KUKA KRL program: EPS_2_251806_MH48A_A_20260213065146.src

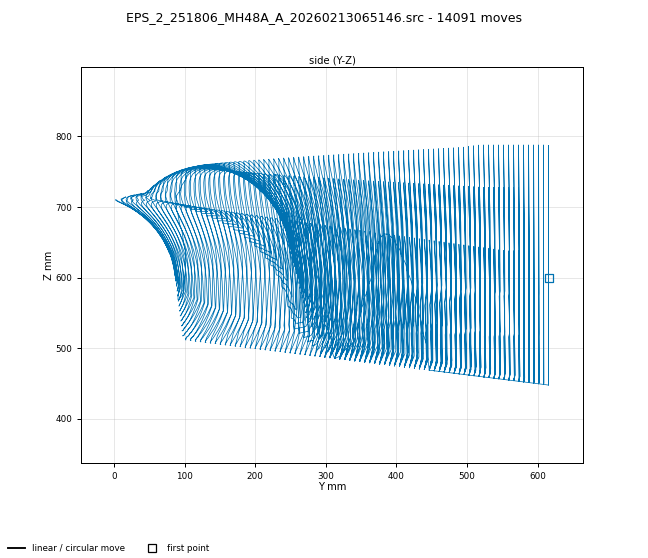
[picture p0: tool path of EPS_2_251806_MH48A_A_20260213065146.src, 14091 of 14093 moves have a stored position in this frame; points joined in program order, loops and branches not executed]
&ACCESS RVP
&REL 4
&COMMENT QRS 19112012
&PARAM EDITMASK = *
DEF PART()
EXT BAS (BAS_COMMAND :IN,REAL :IN )
INT I
BAS (#INITMOV,0 )

;KUKA QRS Post kuka4.cps  Date:22-06-2017 !

File_ID=3035

QRS_PRE_INIT()

;Init var - Until changes are made in qrs_pre_init
Outlet_Square_prg=0
Inlet_1_Square_prg=0
Inlet_2_Square_prg=0
Inlet_3_Square_prg=0
Inlet_4_Square_prg=0
Inlet_5_Square_prg=0

Outlet_1={X 0.000, Y 519.160, Z 687.500, B 0.000, E1 0.000 }
Inlet_1={X 0.000, Y 553.380, Z 207.500, B 0.000, E1 194.000 }
Inlet_2={X 0.000, Y 523.440, Z 627.500, B 0.000, E1 257.000 }
Outlet_1_type=201
Inlet_1_type=201
Inlet_2_type=201
;QRS#1=Sidecore dimensions
;QRS#2=200-8" PVC SDR 35
;QRS#3=200-8" PVC SDR 35
;QRS#4=200-8" PVC SDR 35
;QRS#5=
;QRS#6=
;QRS#7=
;QRS#8=
;QRS#9=12-08 PSX
;QRS#10=12-08 PSX
;QRS#11=12-08 PSX
;QRS#12=
;QRS#13=
;QRS#14=
;QRS#15=
;QRS#16=1220x127x1067 3,5'
;QRS#17=EPS Height
;QRS#18=788
;QRS#19=*
;QRS#20= UPDATED VERSION 22-06-2017
;QRS#21=*
Outlet_Square=0100
Inlet_1_Square=0100
Inlet_2_Square=0100
Inlet_3_Square=0
Inlet_4_Square=0
Inlet_5_Square=0
Mill_Square=1
Outlet_Square_Prg=204
Inlet_1_Square_prg=204
Inlet_2_Square_prg=204

QRS_INIT()

$ADVANCE=5

; T1
PTP {E1 173.589,E2 173.589}
PTP {X 0,Y 615.51,A -85,B 0,C 180,E1 173.589,E2 173.589,E3 0,E4 0,E5 0,E6 0}
QRS_SPEED_INIT()
LIN {X 0,Y 615.51,Z 600,A -85,B 0,C 180,E1 173.589,E2 173.589,E3 0,E4 0,E5 0,E6 0} C_VEL
LIN {X 0,Y 615.51,Z 457.871,A -85,B 0,C 180,E1 173.589,E2 173.589} C_VEL
LIN {X 0,Y 615.51,Z 449.702,A -85,B 0,C 180,E1 173.589,E2 173.589} C_VEL
LIN {X 0,Y 615.493,Z 447.702,A -85,B 0,C 180,E1 173.404,E2 173.404} C_VEL
LIN {X 0,Y 615.484,Z 447.686,A -85,B 0,C 180,E1 170.801,E2 170.801} C_VEL
LIN {X 0,Y 615.449,Z 447.691,A -85,B 0,C 180,E1 168.139,E2 168.139} C_VEL
LIN {X 0,Y 615.487,Z 447.699,A -85,B 0,C 180,E1 165.451,E2 165.451} C_VEL
LIN {X 0,Y 615.488,Z 447.685,A -85,B 0,C 180,E1 162.73,E2 162.73} C_VEL
LIN {X 0,Y 615.482,Z 447.685,A -85,B 0,C 180,E1 160.662,E2 160.662} C_VEL
LIN {X 0,Y 615.478,Z 447.685,A -85,B 0,C 180,E1 158.568,E2 158.568} C_VEL
LIN {X 0,Y 615.456,Z 447.69,A -85,B 0,C 180,E1 155.994,E2 155.994} C_VEL
LIN {X 0,Y 615.473,Z 447.695,A -85,B 0,C 180,E1 153.556,E2 153.556} C_VEL
LIN {X 0,Y 615.485,Z 447.685,A -85,B 0,C 180,E1 150.594,E2 150.594} C_VEL
LIN {X 0,Y 615.469,Z 447.686,A -85,B 0,C 180,E1 148.314,E2 148.314} C_VEL
LIN {X 0,Y 615.457,Z 447.689,A -85,B 0,C 180,E1 145.976,E2 145.976} C_VEL
LIN {X 0,Y 615.491,Z 447.698,A -85,B 0,C 180,E1 143.061,E2 143.061} C_VEL
LIN {X 0,Y 615.472,Z 447.685,A -85,B 0,C 180,E1 140.249,E2 140.249} C_VEL
LIN {X 0,Y 615.466,Z 447.692,A -85,B 0,C 180,E1 137.645,E2 137.645} C_VEL
LIN {X 0,Y 615.492,Z 447.695,A -85,B 0,C 180,E1 134.932,E2 134.932} C_VEL
LIN {X 0,Y 615.487,Z 447.683,A -85,B 0,C 180,E1 132.351,E2 132.351} C_VEL
LIN {X 0,Y 615.465,Z 447.689,A -85,B 0,C 180,E1 129.75,E2 129.75} C_VEL
LIN {X 0,Y 615.494,Z 447.697,A -85,B 0,C 180,E1 126.938,E2 126.938} C_VEL
LIN {X 0,Y 615.472,Z 447.685,A -85,B 0,C 180,E1 124.021,E2 124.021} C_VEL
LIN {X 0,Y 615.468,Z 447.688,A -85,B 0,C 180,E1 121.685,E2 121.685} C_VEL
LIN {X 0,Y 615.475,Z 447.692,A -85,B 0,C 180,E1 119.405,E2 119.405} C_VEL
LIN {X 0,Y 615.492,Z 447.685,A -85,B 0,C 180,E1 116.442,E2 116.442} C_VEL
LIN {X 0,Y 615.479,Z 447.683,A -85,B 0,C 180,E1 114.007,E2 114.007} C_VEL
LIN {X 0,Y 615.476,Z 447.69,A -85,B 0,C 180,E1 111.431,E2 111.431} C_VEL
LIN {X 0,Y 615.488,Z 447.691,A -85,B 0,C 180,E1 108.606,E2 108.606} C_VEL
LIN {X 0,Y 615.479,Z 447.683,A -85,B 0,C 180,E1 105.904,E2 105.904} C_VEL
LIN {X 0,Y 615.487,Z 447.692,A -85,B 0,C 180,E1 103.2,E2 103.2} C_VEL
LIN {X 0,Y 615.487,Z 447.691,A -85,B 0,C 180,E1 100.526,E2 100.526} C_VEL
LIN {X 0,Y 615.483,Z 447.682,A -85,B 0,C 180,E1 97.874,E2 97.874} C_VEL
LIN {X 0,Y 615.479,Z 447.691,A -85,B 0,C 180,E1 95.24,E2 95.24} C_VEL
LIN {X 0,Y 615.486,Z 447.696,A -85,B 0,C 180,E1 92.617,E2 92.617} C_VEL
LIN {X 0,Y 615.487,Z 447.682,A -85,B 0,C 180,E1 89.999,E2 89.999} C_VEL
LIN {X 0,Y 615.498,Z 447.858,A -85,B 0,C 180,E1 88.69,E2 88.69} C_VEL
LIN {X 0,Y 615.497,Z 448.887,A -85,B 0,C 180,E1 88.568,E2 88.568} C_VEL
LIN {X 0,Y 615.498,Z 534.909,A -85,B 0,C 180,E1 87.524,E2 87.524} C_VEL
LIN {X 0,Y 615.498,Z 548.363,A -85,B 0,C 180,E1 87.217,E2 87.217} C_VEL
LIN {X 0,Y 615.499,Z 560.522,A -85,B 0,C 180,E1 86.808,E2 86.808} C_VEL
LIN {X 0,Y 615.497,Z 571.457,A -85,B 0,C 180,E1 86.316,E2 86.316} C_VEL
LIN {X 0,Y 615.491,Z 582.851,A -85,B 0,C 180,E1 85.661,E2 85.661} C_VEL
LIN {X 0,Y 615.498,Z 593.126,A -85,B 0,C 180,E1 84.922,E2 84.922} C_VEL
LIN {X 0,Y 615.5,Z 602.443,A -85,B 0,C 180,E1 84.101,E2 84.101} C_VEL
LIN {X 0,Y 615.496,Z 611.559,A -85,B 0,C 180,E1 83.098,E2 83.098} C_VEL
LIN {X 0,Y 615.496,Z 618.714,A -85,B 0,C 180,E1 82.123,E2 82.123} C_VEL
LIN {X 0,Y 615.496,Z 624.559,A -85,B 0,C 180,E1 81.132,E2 81.132} C_VEL
LIN {X 0,Y 615.497,Z 629.171,A -85,B 0,C 180,E1 80.137,E2 80.137} C_VEL
LIN {X 0,Y 615.495,Z 632.785,A -85,B 0,C 180,E1 79.107,E2 79.107} C_VEL
LIN {X 0,Y 615.496,Z 635.187,A -85,B 0,C 180,E1 78.138,E2 78.138} C_VEL
LIN {X 0,Y 615.495,Z 636.338,A -85,B 0,C 180,E1 77.469,E2 77.469} C_VEL
LIN {X 0,Y 615.496,Z 637.354,A -85,B 0,C 180,E1 76.125,E2 76.125} C_VEL
LIN {X 0,Y 615.497,Z 637.271,A -85,B 0,C 180,E1 75.45,E2 75.45} C_VEL
LIN {X 0,Y 615.496,Z 636.73,A -85,B 0,C 180,E1 74.773,E2 74.773} C_VEL
LIN {X 0,Y 615.494,Z 634.742,A -85,B 0,C 180,E1 73.566,E2 73.566} C_VEL
LIN {X 0,Y 615.496,Z 631.451,A -85,B 0,C 180,E1 72.386,E2 72.386} C_VEL
LIN {X 0,Y 615.497,Z 627.367,A -85,B 0,C 180,E1 71.353,E2 71.353} C_VEL
LIN {X 0,Y 615.497,Z 620.936,A -85,B 0,C 180,E1 70.141,E2 70.141} C_VEL
LIN {X 0,Y 615.497,Z 613.795,A -85,B 0,C 180,E1 69.094,E2 69.094} C_VEL
LIN {X 0,Y 615.499,Z 606.395,A -85,B 0,C 180,E1 68.216,E2 68.216} C_VEL
LIN {X 0,Y 615.5,Z 598.08,A -85,B 0,C 180,E1 67.403,E2 67.403} C_VEL
LIN {X 0,Y 615.5,Z 588.295,A -85,B 0,C 180,E1 66.621,E2 66.621} C_VEL
LIN {X 0,Y 615.488,Z 577.552,A -85,B 0,C 180,E1 65.925,E2 65.925} C_VEL
LIN {X 0,Y 615.499,Z 565.779,A -85,B 0,C 180,E1 65.323,E2 65.323} C_VEL
LIN {X 0,Y 615.498,Z 553.895,A -85,B 0,C 180,E1 64.863,E2 64.863} C_VEL
LIN {X 0,Y 615.499,Z 540.76,A -85,B 0,C 180,E1 64.501,E2 64.501} C_VEL
LIN {X 0,Y 615.494,Z 528.044,A -85,B 0,C 180,E1 64.284,E2 64.284} C_VEL
LIN {X 0,Y 615.496,Z 449.024,A -85,B 0,C 180,E1 63.348,E2 63.348} C_VEL
LIN {X 0,Y 615.498,Z 447.914,A -85,B 0,C 180,E1 63.236,E2 63.236} C_VEL
LIN {X 0,Y 615.493,Z 447.694,A -85,B 0,C 180,E1 61.341,E2 61.341} C_VEL
LIN {X 0,Y 615.495,Z 447.693,A -85,B 0,C 180,E1 58.912,E2 58.912} C_VEL
LIN {X 0,Y 615.473,Z 447.687,A -85,B 0,C 180,E1 56.468,E2 56.468} C_VEL
LIN {X 0,Y 615.465,Z 447.687,A -85,B 0,C 180,E1 54.169,E2 54.169} C_VEL
LIN {X 0,Y 615.471,Z 447.686,A -85,B 0,C 180,E1 51.929,E2 51.929} C_VEL
LIN {X 0,Y 615.495,Z 447.692,A -85,B 0,C 180,E1 49.393,E2 49.393} C_VEL
LIN {X 0,Y 615.499,Z 447.687,A -85,B 0,C 180,E1 46.755,E2 46.755} C_VEL
LIN {X 0,Y 615.464,Z 447.688,A -85,B 0,C 180,E1 43.994,E2 43.994} C_VEL
LIN {X 0,Y 615.491,Z 447.699,A -85,B 0,C 180,E1 41.094,E2 41.094} C_VEL
LIN {X 0,Y 615.486,Z 447.694,A -85,B 0,C 180,E1 38.904,E2 38.904} C_VEL
LIN {X 0,Y 615.473,Z 447.686,A -85,B 0,C 180,E1 36.425,E2 36.425} C_VEL
LIN {X 0,Y 615.498,Z 447.832,A -85,B 0,C 180,E1 35.113,E2 35.113} C_VEL
LIN {X 0,Y 615.498,Z 452.891,A -85,B 0,C 180,E1 34.36,E2 34.36} C_VEL
LIN {X 0,Y 615.491,Z 473.395,A -85,B 0,C 180,E1 31.535,E2 31.535} C_VEL
LIN {X 0,Y 615.491,Z 494.595,A -85,B 0,C 180,E1 28.658,E2 28.658} C_VEL
LIN {X 0,Y 615.486,Z 515.486,A -85,B 0,C 180,E1 25.874,E2 25.874} C_VEL
LIN {X 0,Y 615.491,Z 517.349,A -85,B 0,C 180,E1 25.806,E2 25.806} C_VEL
LIN {X 0,Y 615.495,Z 624.013,A -85,B 0,C 180,E1 24.541,E2 24.541} C_VEL
LIN {X 0,Y 615.498,Z 637.597,A -85,B 0,C 180,E1 24.238,E2 24.238} C_VEL
LIN {X 0,Y 615.497,Z 649.703,A -85,B 0,C 180,E1 23.839,E2 23.839} C_VEL
LIN {X 0,Y 615.494,Z 661.987,A -85,B 0,C 180,E1 23.288,E2 23.288} C_VEL
LIN {X 0,Y 615.497,Z 673.863,A -85,B 0,C 180,E1 22.594,E2 22.594} C_VEL
LIN {X 0,Y 615.498,Z 683.775,A -85,B 0,C 180,E1 21.871,E2 21.871} C_VEL
LIN {X 0,Y 615.499,Z 692.646,A -85,B 0,C 180,E1 21.08,E2 21.08} C_VEL
LIN {X 0,Y 615.498,Z 701.024,A -85,B 0,C 180,E1 20.163,E2 20.163} C_VEL
LIN {X 0,Y 615.498,Z 708.439,A -85,B 0,C 180,E1 19.164,E2 19.164} C_VEL
LIN {X 0,Y 615.498,Z 713.741,A -85,B 0,C 180,E1 18.281,E2 18.281} C_VEL
LIN {X 0,Y 615.497,Z 718.599,A -85,B 0,C 180,E1 17.27,E2 17.27} C_VEL
LIN {X 0,Y 615.497,Z 721.746,A -85,B 0,C 180,E1 16.432,E2 16.432} C_VEL
LIN {X 0,Y 615.498,Z 724.997,A -85,B 0,C 180,E1 15.226,E2 15.226} C_VEL
LIN {X 0,Y 615.494,Z 726.224,A -85,B 0,C 180,E1 14.549,E2 14.549} C_VEL
LIN {X 0,Y 615.494,Z 726.988,A -85,B 0,C 180,E1 13.874,E2 13.874} C_VEL
LIN {X 0,Y 615.494,Z 727.294,A -85,B 0,C 180,E1 12.53,E2 12.53} C_VEL
LIN {X 0,Y 615.495,Z 726.833,A -85,B 0,C 180,E1 11.86,E2 11.86} C_VEL
LIN {X 0,Y 615.494,Z 725.432,A -85,B 0,C 180,E1 10.888,E2 10.888} C_VEL
LIN {X 0,Y 615.497,Z 721.911,A -85,B 0,C 180,E1 9.53,E2 9.53} C_VEL
LIN {X 0,Y 615.495,Z 718.153,A -85,B 0,C 180,E1 8.536,E2 8.536} C_VEL
LIN {X 0,Y 615.497,Z 713.28,A -85,B 0,C 180,E1 7.545,E2 7.545} C_VEL
LIN {X 0,Y 615.496,Z 707.158,A -85,B 0,C 180,E1 6.556,E2 6.556} C_VEL
LIN {X 0,Y 615.498,Z 699.562,A -85,B 0,C 180,E1 5.569,E2 5.569} C_VEL
LIN {X 0,Y 615.497,Z 690.049,A -85,B 0,C 180,E1 4.584,E2 4.584} C_VEL
LIN {X 0,Y 615.5,Z 680.271,A -85,B 0,C 180,E1 3.764,E2 3.764} C_VEL
LIN {X 0,Y 615.493,Z 669.27,A -85,B 0,C 180,E1 3.027,E2 3.027} C_VEL
LIN {X 0,Y 615.497,Z 658.558,A -85,B 0,C 180,E1 2.454,E2 2.454} C_VEL
LIN {X 0,Y 615.499,Z 646.783,A -85,B 0,C 180,E1 1.963,E2 1.963} C_VEL
LIN {X 0,Y 615.498,Z 634.795,A -85,B 0,C 180,E1 1.595,E2 1.595} C_VEL
LIN {X 0,Y 615.499,Z 622.775,A -85,B 0,C 180,E1 1.349,E2 1.349} C_VEL
LIN {X 0,Y 615.493,Z 516.279,A -85,B 0,C 180,E1 0.082,E2 0.082} C_VEL
LIN {X 0,Y 615.486,Z 515.176,A -85,B 0,C 180,E1 0,E2 0} C_VEL
LIN {X 0,Y 615.485,Z 494.453,A -85,B 0,C 180,E1 -2.782,E2 -2.782} C_VEL
LIN {X 0,Y 615.499,Z 473.986,A -85,B 0,C 180,E1 -5.57,E2 -5.57} C_VEL
LIN {X 0,Y 615.496,Z 453.734,A -85,B 0,C 180,E1 -8.371,E2 -8.371} C_VEL
LIN {X 0,Y 615.498,Z 447.975,A -85,B 0,C 180,E1 -9.199,E2 -9.199} C_VEL
LIN {X 0,Y 615.461,Z 447.692,A -85,B 0,C 180,E1 -9.863,E2 -9.863} C_VEL
LIN {X 0,Y 615.465,Z 447.691,A -85,B 0,C 180,E1 -11.861,E2 -11.861} C_VEL
LIN {X 0,Y 615.46,Z 447.69,A -85,B 0,C 180,E1 -13.92,E2 -13.92} C_VEL
LIN {X 0,Y 615.443,Z 447.695,A -85,B 0,C 180,E1 -16.415,E2 -16.415} C_VEL
LIN {X 0,Y 615.451,Z 447.698,A -85,B 0,C 180,E1 -18.647,E2 -18.647} C_VEL
LIN {X 0,Y 615.496,Z 447.688,A -85,B 0,C 180,E1 -21.432,E2 -21.432} C_VEL
LIN {X 0,Y 615.461,Z 447.691,A -85,B 0,C 180,E1 -24.273,E2 -24.273} C_VEL
LIN {X 0,Y 615.466,Z 447.694,A -85,B 0,C 180,E1 -26.445,E2 -26.445} C_VEL
LIN {X 0,Y 615.481,Z 447.698,A -85,B 0,C 180,E1 -28.659,E2 -28.659} C_VEL
LIN {X 0,Y 615.493,Z 447.691,A -85,B 0,C 180,E1 -31.085,E2 -31.085} C_VEL
LIN {X 0,Y 615.479,Z 447.687,A -85,B 0,C 180,E1 -34.023,E2 -34.023} C_VEL
LIN {X 0,Y 615.484,Z 447.696,A -85,B 0,C 180,E1 -36.425,E2 -36.425} C_VEL
LIN {X 0,Y 615.484,Z 447.689,A -85,B 0,C 180,E1 -39.061,E2 -39.061} C_VEL
LIN {X 0,Y 615.498,Z 447.68,A -85,B 0,C 180,E1 -41.473,E2 -41.473} C_VEL
LIN {X 0,Y 615.487,Z 447.692,A -85,B 0,C 180,E1 -44.15,E2 -44.15} C_VEL
LIN {X 0,Y 615.471,Z 447.69,A -85,B 0,C 180,E1 -46.955,E2 -46.955} C_VEL
LIN {X 0,Y 615.485,Z 447.683,A -85,B 0,C 180,E1 -49.392,E2 -49.392} C_VEL
LIN {X 0,Y 615.495,Z 447.691,A -85,B 0,C 180,E1 -51.988,E2 -51.988} C_VEL
LIN {X 0,Y 615.481,Z 447.698,A -85,B 0,C 180,E1 -54.383,E2 -54.383} C_VEL
LIN {X 0,Y 615.452,Z 447.694,A -85,B 0,C 180,E1 -56.761,E2 -56.761} C_VEL
LIN {X 0,Y 615.448,Z 447.692,A -85,B 0,C 180,E1 -59.077,E2 -59.077} C_VEL
LIN {X 0,Y 615.482,Z 447.689,A -85,B 0,C 180,E1 -61.551,E2 -61.551} C_VEL
LIN {X 0,Y 615.494,Z 447.895,A -85,B 0,C 180,E1 -64.102,E2 -64.102} C_VEL
LIN {X 0,Y 615.495,Z 451.94,A -85,B 0,C 180,E1 -64.574,E2 -64.574} C_VEL
LIN {X 0,Y 615.497,Z 478.617,A -85,B 0,C 180,E1 -67.405,E2 -67.405} C_VEL
LIN {X 0,Y 615.489,Z 504.931,A -85,B 0,C 180,E1 -70.14,E2 -70.14} C_VEL
LIN {X 0,Y 615.445,Z 530.237,A -85,B 0,C 180,E1 -72.727,E2 -72.727} C_VEL
LIN {X 0,Y 615.481,Z 555.512,A -85,B 0,C 180,E1 -75.281,E2 -75.281} C_VEL
LIN {X 0,Y 615.493,Z 573.822,A -85,B 0,C 180,E1 -77.092,E2 -77.092} C_VEL
LIN {X 0,Y 615.489,Z 683.773,A -85,B 0,C 180,E1 -78.41,E2 -78.41} C_VEL
LIN {X 0,Y 615.499,Z 696.305,A -85,B 0,C 180,E1 -78.681,E2 -78.681} C_VEL
LIN {X 0,Y 615.496,Z 709.501,A -85,B 0,C 180,E1 -79.109,E2 -79.109} C_VEL
LIN {X 0,Y 615.491,Z 721.457,A -85,B 0,C 180,E1 -79.638,E2 -79.638} C_VEL
LIN {X 0,Y 615.488,Z 732.979,A -85,B 0,C 180,E1 -80.303,E2 -80.303} C_VEL
LIN {X 0,Y 615.499,Z 743.328,A -85,B 0,C 180,E1 -81.049,E2 -81.049} C_VEL
LIN {X 0,Y 615.497,Z 751.801,A -85,B 0,C 180,E1 -81.793,E2 -81.793} C_VEL
LIN {X 0,Y 615.498,Z 759.597,A -85,B 0,C 180,E1 -82.619,E2 -82.619} C_VEL
LIN {X 0,Y 615.497,Z 767.196,A -85,B 0,C 180,E1 -83.607,E2 -83.607} C_VEL
LIN {X 0,Y 615.498,Z 774.199,A -85,B 0,C 180,E1 -84.758,E2 -84.758} C_VEL
LIN {X 0,Y 615.494,Z 778.847,A -85,B 0,C 180,E1 -85.743,E2 -85.743} C_VEL
LIN {X 0,Y 615.494,Z 782.395,A -85,B 0,C 180,E1 -86.726,E2 -86.726} C_VEL
LIN {X 0,Y 615.497,Z 784.23,A -85,B 0,C 180,E1 -87.381,E2 -87.381} C_VEL
LIN {X 0,Y 615.498,Z 785.606,A -85,B 0,C 180,E1 -88.036,E2 -88.036} C_VEL
LIN {X 0,Y 615.496,Z 787.173,A -85,B 0,C 180,E1 -89.345,E2 -89.345} C_VEL
LIN {X 0,Y 615.494,Z 787.389,A -85,B 0,C 180,E1 -89.999,E2 -89.999} C_VEL
LIN {X 0,Y 615.495,Z 786.581,A -85,B 0,C 180,E1 -91.307,E2 -91.307} C_VEL
LIN {X 0,Y 615.498,Z 785.61,A -85,B 0,C 180,E1 -91.962,E2 -91.962} C_VEL
LIN {X 0,Y 615.497,Z 784.236,A -85,B 0,C 180,E1 -92.617,E2 -92.617} C_VEL
LIN {X 0,Y 615.496,Z 781.353,A -85,B 0,C 180,E1 -93.599,E2 -93.599} C_VEL
LIN {X 0,Y 615.498,Z 777.446,A -85,B 0,C 180,E1 -94.583,E2 -94.583} C_VEL
LIN {X 0,Y 615.499,Z 772.411,A -85,B 0,C 180,E1 -95.569,E2 -95.569} C_VEL
LIN {X 0,Y 615.497,Z 765.87,A -85,B 0,C 180,E1 -96.583,E2 -96.583} C_VEL
LIN {X 0,Y 615.497,Z 758.144,A -85,B 0,C 180,E1 -97.544,E2 -97.544} C_VEL
LIN {X 0,Y 615.498,Z 750.057,A -85,B 0,C 180,E1 -98.37,E2 -98.37} C_VEL
LIN {X 0,Y 615.499,Z 740.183,A -85,B 0,C 180,E1 -99.197,E2 -99.197} C_VEL
LIN {X 0,Y 615.489,Z 729.001,A -85,B 0,C 180,E1 -99.944,E2 -99.944} C_VEL
LIN {X 0,Y 615.491,Z 718.047,A -85,B 0,C 180,E1 -100.526,E2 -100.526} C_VEL
LIN {X 0,Y 615.499,Z 705.434,A -85,B 0,C 180,E1 -101.042,E2 -101.042} C_VEL
LIN {X 0,Y 615.498,Z 693.116,A -85,B 0,C 180,E1 -101.4,E2 -101.4} C_VEL
LIN {X 0,Y 615.488,Z 679.554,A -85,B 0,C 180,E1 -101.651,E2 -101.651} C_VEL
LIN {X 0,Y 615.492,Z 573.891,A -85,B 0,C 180,E1 -102.906,E2 -102.906} C_VEL
LIN {X 0,Y 615.448,Z 550.6,A -85,B 0,C 180,E1 -105.226,E2 -105.226} C_VEL
LIN {X 0,Y 615.498,Z 523.74,A -85,B 0,C 180,E1 -107.955,E2 -107.955} C_VEL
LIN {X 0,Y 615.479,Z 496.849,A -85,B 0,C 180,E1 -110.73,E2 -110.73} C_VEL
LIN {X 0,Y 615.454,Z 473.315,A -85,B 0,C 180,E1 -113.2,E2 -113.2} C_VEL
LIN {X 0,Y 615.494,Z 449.781,A -85,B 0,C 180,E1 -115.714,E2 -115.714} C_VEL
LIN {X 0,Y 615.495,Z 447.941,A -85,B 0,C 180,E1 -115.941,E2 -115.941} C_VEL
LIN {X 0,Y 615.425,Z 447.696,A -85,B 0,C 180,E1 -117.179,E2 -117.179} C_VEL
LIN {X 0,Y 615.457,Z 447.699,A -85,B 0,C 180,E1 -119.789,E2 -119.789} C_VEL
LIN {X 0,Y 615.485,Z 447.692,A -85,B 0,C 180,E1 -122.456,E2 -122.456} C_VEL
LIN {X 0,Y 615.446,Z 447.693,A -85,B 0,C 180,E1 -124.816,E2 -124.816} C_VEL
LIN {X 0,Y 615.428,Z 447.695,A -85,B 0,C 180,E1 -127.245,E2 -127.245} C_VEL
LIN {X 0,Y 615.486,Z 447.7,A -85,B 0,C 180,E1 -130.088,E2 -130.088} C_VEL
LIN {X 0,Y 615.499,Z 447.694,A -85,B 0,C 180,E1 -132.35,E2 -132.35} C_VEL
LIN {X 0,Y 615.438,Z 447.693,A -85,B 0,C 180,E1 -135.071,E2 -135.071} C_VEL
LIN {X 0,Y 615.438,Z 447.696,A -85,B 0,C 180,E1 -137.642,E2 -137.642} C_VEL
LIN {X 0,Y 615.496,Z 447.701,A -85,B 0,C 180,E1 -140.25,E2 -140.25} C_VEL
LIN {X 0,Y 615.445,Z 447.692,A -85,B 0,C 180,E1 -143.066,E2 -143.066} C_VEL
LIN {X 0,Y 615.436,Z 447.693,A -85,B 0,C 180,E1 -145.304,E2 -145.304} C_VEL
LIN {X 0,Y 615.438,Z 447.696,A -85,B 0,C 180,E1 -147.674,E2 -147.674} C_VEL
LIN {X 0,Y 615.481,Z 447.699,A -85,B 0,C 180,E1 -150.203,E2 -150.203} C_VEL
LIN {X 0,Y 615.467,Z 447.69,A -85,B 0,C 180,E1 -152.955,E2 -152.955} C_VEL
LIN {X 0,Y 615.464,Z 447.69,A -85,B 0,C 180,E1 -155.007,E2 -155.007} C_VEL
LIN {X 0,Y 615.453,Z 447.69,A -85,B 0,C 180,E1 -157.154,E2 -157.154} C_VEL
LIN {X 0,Y 615.44,Z 447.692,A -85,B 0,C 180,E1 -159.45,E2 -159.45} C_VEL
LIN {X 0,Y 615.44,Z 447.692,A -85,B 0,C 180,E1 -161.403,E2 -161.403} C_VEL
LIN {X 0,Y 615.44,Z 447.693,A -85,B 0,C 180,E1 -163.578,E2 -163.578} C_VEL
LIN {X 0,Y 615.46,Z 447.698,A -85,B 0,C 180,E1 -166.125,E2 -166.125} C_VEL
LIN {X 0,Y 615.471,Z 447.688,A -85,B 0,C 180,E1 -169.112,E2 -169.112} C_VEL
LIN {X 0,Y 615.448,Z 447.69,A -85,B 0,C 180,E1 -171.463,E2 -171.463} C_VEL
LIN {X 0,Y 615.447,Z 447.691,A -85,B 0,C 180,E1 -173.443,E2 -173.443} C_VEL
LIN {X 0,Y 615.453,Z 447.689,A -85,B 0,C 180,E1 -175.415,E2 -175.415} C_VEL
LIN {X 0,Y 615.457,Z 447.689,A -85,B 0,C 180,E1 -177.382,E2 -177.382} C_VEL
LIN {X 0,Y 615.462,Z 447.688,A -85,B 0,C 180,E1 -179.345,E2 -179.345} C_VEL
LIN {X 0,Y 615.451,Z 447.693,A -85,B 0,C 180,E1 -181.963,E2 -181.963} C_VEL
LIN {X 0,Y 615.5,Z 447.7,A -85,B 0,C 180,E1 -184.584,E2 -184.584} C_VEL
LIN {X 0,Y 615.493,Z 447.702,A -85,B 0,C 180,E1 -186.596,E2 -186.596} C_VEL
LIN {X 0,Y 614.812,Z 447.834,A -85,B 0,C 180,E1 -187.142,E2 -187.142} C_VEL
LIN {X 0,Y 611.977,Z 448.25,A -85,B 0,C 180,E1 -188.028,E2 -188.028} C_VEL
LIN {X 0,Y 609.582,Z 448.56,A -85,B 0,C 180,E1 -188.74,E2 -188.74} C_VEL
LIN {X 0,Y 608.539,Z 448.678,A -85,B 0,C 180,E1 -189.29,E2 -189.29} C_VEL
LIN {X 0,Y 608.445,Z 448.688,A -85,B 0,C 180,E1 -189.476,E2 -189.476} C_VEL
LIN {X 0,Y 608.435,Z 448.691,A -85,B 0,C 180,E1 -192,E2 -192} C_VEL
LIN {X 0,Y 608.474,Z 448.694,A -85,B 0,C 180,E1 -194.72,E2 -194.72} C_VEL
LIN {X 0,Y 608.443,Z 448.688,A -85,B 0,C 180,E1 -197.477,E2 -197.477} C_VEL
LIN {X 0,Y 608.438,Z 448.689,A -85,B 0,C 180,E1 -199.571,E2 -199.571} C_VEL
LIN {X 0,Y 608.462,Z 448.691,A -85,B 0,C 180,E1 -202.406,E2 -202.406} C_VEL
LIN {X 0,Y 608.445,Z 448.69,A -85,B 0,C 180,E1 -205.301,E2 -205.301} C_VEL
LIN {X 0,Y 608.437,Z 448.689,A -85,B 0,C 180,E1 -207.518,E2 -207.518} C_VEL
LIN {X 0,Y 608.443,Z 448.688,A -85,B 0,C 180,E1 -209.971,E2 -209.971} C_VEL
LIN {X 0,Y 608.452,Z 448.693,A -85,B 0,C 180,E1 -212.524,E2 -212.524} C_VEL
LIN {X 0,Y 608.444,Z 448.691,A -85,B 0,C 180,E1 -215.277,E2 -215.277} C_VEL
LIN {X 0,Y 608.455,Z 448.687,A -85,B 0,C 180,E1 -217.747,E2 -217.747} C_VEL
LIN {X 0,Y 608.436,Z 448.692,A -85,B 0,C 180,E1 -220.33,E2 -220.33} C_VEL
LIN {X 0,Y 608.453,Z 448.696,A -85,B 0,C 180,E1 -222.959,E2 -222.959} C_VEL
LIN {X 0,Y 608.443,Z 448.688,A -85,B 0,C 180,E1 -225.737,E2 -225.737} C_VEL
LIN {X 0,Y 608.449,Z 448.687,A -85,B 0,C 180,E1 -227.94,E2 -227.94} C_VEL
LIN {X 0,Y 608.473,Z 448.691,A -85,B 0,C 180,E1 -230.702,E2 -230.702} C_VEL
LIN {X 0,Y 608.464,Z 448.694,A -85,B 0,C 180,E1 -233.087,E2 -233.087} C_VEL
LIN {X 0,Y 608.465,Z 448.687,A -85,B 0,C 180,E1 -235.532,E2 -235.532} C_VEL
LIN {X 0,Y 608.465,Z 448.685,A -85,B 0,C 180,E1 -237.907,E2 -237.907} C_VEL
LIN {X 0,Y 608.451,Z 448.688,A -85,B 0,C 180,E1 -240.221,E2 -240.221} C_VEL
LIN {X 0,Y 608.482,Z 448.69,A -85,B 0,C 180,E1 -242.792,E2 -242.792} C_VEL
LIN {X 0,Y 608.474,Z 448.684,A -85,B 0,C 180,E1 -245.848,E2 -245.848} C_VEL
LIN {X 0,Y 608.463,Z 448.686,A -85,B 0,C 180,E1 -248.31,E2 -248.31} C_VEL
LIN {X 0,Y 608.47,Z 448.692,A -85,B 0,C 180,E1 -251.283,E2 -251.283} C_VEL
LIN {X 0,Y 608.457,Z 448.687,A -85,B 0,C 180,E1 -253.907,E2 -253.907} C_VEL
LIN {X 0,Y 608.463,Z 448.689,A -85,B 0,C 180,E1 -256.645,E2 -256.645} C_VEL
LIN {X 0,Y 608.468,Z 448.692,A -85,B 0,C 180,E1 -259.351,E2 -259.351} C_VEL
LIN {X 0,Y 608.475,Z 448.684,A -85,B 0,C 180,E1 -262.034,E2 -262.034} C_VEL
LIN {X 0,Y 608.46,Z 448.689,A -85,B 0,C 180,E1 -264.699,E2 -264.699} C_VEL
LIN {X 0,Y 608.477,Z 448.692,A -85,B 0,C 180,E1 -267.353,E2 -267.353} C_VEL
LIN {X 0,Y 608.478,Z 448.685,A -85,B 0,C 180,E1 -270.001,E2 -270.001} C_VEL
LIN {X 0,Y 608.499,Z 448.858,A -85,B 0,C 180,E1 -271.201,E2 -271.201} C_VEL
LIN {X 0,Y 608.588,Z 449.873,A -85,B 0,C 180,E1 -271.304,E2 -271.304} C_VEL
LIN {X 0,Y 608.56,Z 534.836,A -85,B 0,C 180,E1 -272.338,E2 -272.338} C_VEL
LIN {X 0,Y 608.55,Z 548.357,A -85,B 0,C 180,E1 -272.649,E2 -272.649} C_VEL
LIN {X 0,Y 608.545,Z 560.563,A -85,B 0,C 180,E1 -273.063,E2 -273.063} C_VEL
LIN {X 0,Y 608.511,Z 571.556,A -85,B 0,C 180,E1 -273.56,E2 -273.56} C_VEL
LIN {X 0,Y 608.504,Z 583.002,A -85,B 0,C 180,E1 -274.224,E2 -274.224} C_VEL
LIN {X 0,Y 608.476,Z 593.34,A -85,B 0,C 180,E1 -274.971,E2 -274.971} C_VEL
LIN {X 0,Y 608.479,Z 602.714,A -85,B 0,C 180,E1 -275.801,E2 -275.801} C_VEL
LIN {X 0,Y 608.46,Z 611.778,A -85,B 0,C 180,E1 -276.8,E2 -276.8} C_VEL
LIN {X 0,Y 608.454,Z 619.116,A -85,B 0,C 180,E1 -277.801,E2 -277.801} C_VEL
LIN {X 0,Y 608.448,Z 624.103,A -85,B 0,C 180,E1 -278.637,E2 -278.637} C_VEL
LIN {X 0,Y 608.43,Z 628.959,A -85,B 0,C 180,E1 -279.643,E2 -279.643} C_VEL
LIN {X 0,Y 608.436,Z 632.692,A -85,B 0,C 180,E1 -280.651,E2 -280.651} C_VEL
LIN {X 0,Y 608.425,Z 634.621,A -85,B 0,C 180,E1 -281.326,E2 -281.326} C_VEL
LIN {X 0,Y 608.44,Z 636.105,A -85,B 0,C 180,E1 -282.001,E2 -282.001} C_VEL
LIN {X 0,Y 608.44,Z 637.766,A -85,B 0,C 180,E1 -283.358,E2 -283.358} C_VEL
LIN {X 0,Y 608.423,Z 638,A -85,B 0,C 180,E1 -284.04,E2 -284.04} C_VEL
LIN {X 0,Y 608.418,Z 637.772,A -85,B 0,C 180,E1 -284.723,E2 -284.723} C_VEL
LIN {X 0,Y 608.418,Z 637.137,A -85,B 0,C 180,E1 -285.408,E2 -285.408} C_VEL
LIN {X 0,Y 608.422,Z 635.209,A -85,B 0,C 180,E1 -286.515,E2 -286.515} C_VEL
LIN {X 0,Y 608.424,Z 632.565,A -85,B 0,C 180,E1 -287.478,E2 -287.478} C_VEL
LIN {X 0,Y 608.431,Z 627.851,A -85,B 0,C 180,E1 -288.706,E2 -288.706} C_VEL
LIN {X 0,Y 608.452,Z 622.474,A -85,B 0,C 180,E1 -289.747,E2 -289.747} C_VEL
LIN {X 0,Y 608.467,Z 615.652,A -85,B 0,C 180,E1 -290.788,E2 -290.788} C_VEL
LIN {X 0,Y 608.455,Z 606.757,A -85,B 0,C 180,E1 -291.871,E2 -291.871} C_VEL
LIN {X 0,Y 608.472,Z 596.837,A -85,B 0,C 180,E1 -292.828,E2 -292.828} C_VEL
LIN {X 0,Y 608.49,Z 586.063,A -85,B 0,C 180,E1 -293.664,E2 -293.664} C_VEL
LIN {X 0,Y 608.513,Z 574.307,A -85,B 0,C 180,E1 -294.383,E2 -294.383} C_VEL
LIN {X 0,Y 608.515,Z 561.742,A -85,B 0,C 180,E1 -294.979,E2 -294.979} C_VEL
LIN {X 0,Y 608.547,Z 548.907,A -85,B 0,C 180,E1 -295.426,E2 -295.426} C_VEL
LIN {X 0,Y 608.57,Z 535.422,A -85,B 0,C 180,E1 -295.741,E2 -295.741} C_VEL
LIN {X 0,Y 608.574,Z 505.219,A -85,B 0,C 180,E1 -296.123,E2 -296.123} C_VEL
LIN {X 0,Y 608.601,Z 449.871,A -85,B 0,C 180,E1 -296.787,E2 -296.787} C_VEL
LIN {X 0,Y 608.484,Z 448.796,A -85,B 0,C 180,E1 -296.907,E2 -296.907} C_VEL
LIN {X 0,Y 608.469,Z 448.693,A -85,B 0,C 180,E1 -299.021,E2 -299.021} C_VEL
LIN {X 0,Y 608.448,Z 448.691,A -85,B 0,C 180,E1 -301.319,E2 -301.319} C_VEL
LIN {X 0,Y 608.448,Z 448.688,A -85,B 0,C 180,E1 -303.732,E2 -303.732} C_VEL
LIN {X 0,Y 608.445,Z 448.689,A -85,B 0,C 180,E1 -306.093,E2 -306.093} C_VEL
LIN {X 0,Y 608.443,Z 448.695,A -85,B 0,C 180,E1 -308.591,E2 -308.591} C_VEL
LIN {X 0,Y 608.46,Z 448.689,A -85,B 0,C 180,E1 -311.342,E2 -311.342} C_VEL
LIN {X 0,Y 608.453,Z 448.687,A -85,B 0,C 180,E1 -313.872,E2 -313.872} C_VEL
LIN {X 0,Y 608.484,Z 448.692,A -85,B 0,C 180,E1 -316.691,E2 -316.691} C_VEL
LIN {X 0,Y 608.461,Z 448.697,A -85,B 0,C 180,E1 -318.824,E2 -318.824} C_VEL
LIN {X 0,Y 608.45,Z 448.688,A -85,B 0,C 180,E1 -321.763,E2 -321.763} C_VEL
LIN {X 0,Y 608.442,Z 448.69,A -85,B 0,C 180,E1 -323.956,E2 -323.956} C_VEL
LIN {X 0,Y 608.489,Z 448.849,A -85,B 0,C 180,E1 -324.785,E2 -324.785} C_VEL
LIN {X 0,Y 608.55,Z 459.678,A -85,B 0,C 180,E1 -326.335,E2 -326.335} C_VEL
LIN {X 0,Y 608.517,Z 480.832,A -85,B 0,C 180,E1 -329.266,E2 -329.266} C_VEL
LIN {X 0,Y 608.504,Z 500.317,A -85,B 0,C 180,E1 -331.924,E2 -331.924} C_VEL
LIN {X 0,Y 608.48,Z 515.928,A -85,B 0,C 180,E1 -334.003,E2 -334.003} C_VEL
LIN {X 0,Y 608.595,Z 520.305,A -85,B 0,C 180,E1 -334.081,E2 -334.081} C_VEL
LIN {X 0,Y 608.544,Z 623.822,A -85,B 0,C 180,E1 -335.319,E2 -335.319} C_VEL
LIN {X 0,Y 608.557,Z 637.32,A -85,B 0,C 180,E1 -335.62,E2 -335.62} C_VEL
LIN {X 0,Y 608.543,Z 650.062,A -85,B 0,C 180,E1 -336.044,E2 -336.044} C_VEL
LIN {X 0,Y 608.512,Z 660.711,A -85,B 0,C 180,E1 -336.519,E2 -336.519} C_VEL
LIN {X 0,Y 608.491,Z 672.257,A -85,B 0,C 180,E1 -337.174,E2 -337.174} C_VEL
LIN {X 0,Y 608.498,Z 683.113,A -85,B 0,C 180,E1 -337.953,E2 -337.953} C_VEL
LIN {X 0,Y 608.477,Z 693.12,A -85,B 0,C 180,E1 -338.842,E2 -338.842} C_VEL
LIN {X 0,Y 608.46,Z 701.171,A -85,B 0,C 180,E1 -339.726,E2 -339.726} C_VEL
LIN {X 0,Y 608.442,Z 708.973,A -85,B 0,C 180,E1 -340.78,E2 -340.78} C_VEL
LIN {X 0,Y 608.446,Z 715.145,A -85,B 0,C 180,E1 -341.828,E2 -341.828} C_VEL
LIN {X 0,Y 608.456,Z 719.922,A -85,B 0,C 180,E1 -342.87,E2 -342.87} C_VEL
LIN {X 0,Y 608.433,Z 723.493,A -85,B 0,C 180,E1 -343.906,E2 -343.906} C_VEL
LIN {X 0,Y 608.422,Z 725.248,A -85,B 0,C 180,E1 -344.593,E2 -344.593} C_VEL
LIN {X 0,Y 608.418,Z 726.566,A -85,B 0,C 180,E1 -345.278,E2 -345.278} C_VEL
LIN {X 0,Y 608.446,Z 727.501,A -85,B 0,C 180,E1 -345.995,E2 -345.995} C_VEL
LIN {X 0,Y 608.44,Z 727.912,A -85,B 0,C 180,E1 -346.643,E2 -346.643} C_VEL
LIN {X 0,Y 608.44,Z 727.578,A -85,B 0,C 180,E1 -348,E2 -348} C_VEL
LIN {X 0,Y 608.451,Z 726.159,A -85,B 0,C 180,E1 -349.057,E2 -349.057} C_VEL
LIN {X 0,Y 608.43,Z 722.949,A -85,B 0,C 180,E1 -350.358,E2 -350.358} C_VEL
LIN {X 0,Y 608.428,Z 719.316,A -85,B 0,C 180,E1 -351.364,E2 -351.364} C_VEL
LIN {X 0,Y 608.451,Z 714.571,A -85,B 0,C 180,E1 -352.367,E2 -352.367} C_VEL
LIN {X 0,Y 608.447,Z 707.698,A -85,B 0,C 180,E1 -353.499,E2 -353.499} C_VEL
LIN {X 0,Y 608.462,Z 699.778,A -85,B 0,C 180,E1 -354.532,E2 -354.532} C_VEL
LIN {X 0,Y 608.474,Z 690.172,A -85,B 0,C 180,E1 -355.529,E2 -355.529} C_VEL
LIN {X 0,Y 608.48,Z 680.305,A -85,B 0,C 180,E1 -356.358,E2 -356.358} C_VEL
LIN {X 0,Y 608.503,Z 669.192,A -85,B 0,C 180,E1 -357.104,E2 -357.104} C_VEL
LIN {X 0,Y 608.513,Z 658.384,A -85,B 0,C 180,E1 -357.684,E2 -357.684} C_VEL
LIN {X 0,Y 608.54,Z 646.491,A -85,B 0,C 180,E1 -358.18,E2 -358.18} C_VEL
LIN {X 0,Y 608.555,Z 634.267,A -85,B 0,C 180,E1 -358.553,E2 -358.553} C_VEL
LIN {X 0,Y 608.548,Z 621.805,A -85,B 0,C 180,E1 -358.801,E2 -358.801} C_VEL
LIN {X 0,Y 608.546,Z 516.463,A -85,B 0,C 180,E1 -360.062,E2 -360.062} C_VEL
LIN {X 0,Y 608.457,Z 515.193,A -85,B 0,C 180,E1 -360.166,E2 -360.166} C_VEL
LIN {X 0,Y 608.492,Z 495.654,A -85,B 0,C 180,E1 -362.814,E2 -362.814} C_VEL
LIN {X 0,Y 608.553,Z 475.135,A -85,B 0,C 180,E1 -365.634,E2 -365.634} C_VEL
LIN {X 0,Y 608.566,Z 454.863,A -85,B 0,C 180,E1 -368.467,E2 -368.467} C_VEL
LIN {X 0,Y 608.498,Z 448.826,A -85,B 0,C 180,E1 -369.348,E2 -369.348} C_VEL
LIN {X 0,Y 608.44,Z 448.69,A -85,B 0,C 180,E1 -372,E2 -372} C_VEL
LIN {X 0,Y 608.427,Z 448.691,A -85,B 0,C 180,E1 -374.039,E2 -374.039} C_VEL
LIN {X 0,Y 608.416,Z 448.694,A -85,B 0,C 180,E1 -376.51,E2 -376.51} C_VEL
LIN {X 0,Y 608.447,Z 448.695,A -85,B 0,C 180,E1 -378.87,E2 -378.87} C_VEL
LIN {X 0,Y 608.461,Z 448.688,A -85,B 0,C 180,E1 -381.692,E2 -381.692} C_VEL
LIN {X 0,Y 608.446,Z 448.693,A -85,B 0,C 180,E1 -384.572,E2 -384.572} C_VEL
LIN {X 0,Y 608.487,Z 448.688,A -85,B 0,C 180,E1 -387.207,E2 -387.207} C_VEL
LIN {X 0,Y 608.464,Z 448.686,A -85,B 0,C 180,E1 -389.97,E2 -389.97} C_VEL
LIN {X 0,Y 608.458,Z 448.694,A -85,B 0,C 180,E1 -392.521,E2 -392.521} C_VEL
LIN {X 0,Y 608.453,Z 448.689,A -85,B 0,C 180,E1 -395.277,E2 -395.277} C_VEL
LIN {X 0,Y 608.47,Z 448.686,A -85,B 0,C 180,E1 -397.746,E2 -397.746} C_VEL
LIN {X 0,Y 608.453,Z 448.694,A -85,B 0,C 180,E1 -400.328,E2 -400.328} C_VEL
LIN {X 0,Y 608.473,Z 448.685,A -85,B 0,C 180,E1 -403.308,E2 -403.308} C_VEL
LIN {X 0,Y 608.474,Z 448.691,A -85,B 0,C 180,E1 -406.13,E2 -406.13} C_VEL
LIN {X 0,Y 608.44,Z 448.692,A -85,B 0,C 180,E1 -408.821,E2 -408.821} C_VEL
LIN {X 0,Y 608.472,Z 448.687,A -85,B 0,C 180,E1 -411.76,E2 -411.76} C_VEL
LIN {X 0,Y 608.433,Z 448.692,A -85,B 0,C 180,E1 -414.721,E2 -414.721} C_VEL
LIN {X 0,Y 608.463,Z 448.688,A -85,B 0,C 180,E1 -417.478,E2 -417.478} C_VEL
LIN {X 0,Y 608.468,Z 448.694,A -85,B 0,C 180,E1 -420.219,E2 -420.219} C_VEL
LIN {X 0,Y 608.418,Z 448.694,A -85,B 0,C 180,E1 -422.804,E2 -422.804} C_VEL
LIN {X 0,Y 608.499,Z 448.815,A -85,B 0,C 180,E1 -423.897,E2 -423.897} C_VEL
LIN {X 0,Y 608.752,Z 451.506,A -85,B 0,C 180,E1 -424.225,E2 -424.225} C_VEL
LIN {X 0,Y 608.631,Z 476.239,A -85,B 0,C 180,E1 -426.882,E2 -426.882} C_VEL
LIN {X 0,Y 608.611,Z 503.243,A -85,B 0,C 180,E1 -429.73,E2 -429.73} C_VEL
LIN {X 0,Y 608.525,Z 530.247,A -85,B 0,C 180,E1 -432.525,E2 -432.525} C_VEL
LIN {X 0,Y 608.499,Z 555.563,A -85,B 0,C 180,E1 -435.108,E2 -435.108} C_VEL
LIN {X 0,Y 608.53,Z 573.861,A -85,B 0,C 180,E1 -436.941,E2 -436.941} C_VEL
LIN {X 0,Y 608.541,Z 683.891,A -85,B 0,C 180,E1 -438.275,E2 -438.275} C_VEL
LIN {X 0,Y 608.547,Z 697.179,A -85,B 0,C 180,E1 -438.571,E2 -438.571} C_VEL
LIN {X 0,Y 608.545,Z 710.321,A -85,B 0,C 180,E1 -439.009,E2 -439.009} C_VEL
LIN {X 0,Y 608.509,Z 721.615,A -85,B 0,C 180,E1 -439.518,E2 -439.518} C_VEL
LIN {X 0,Y 608.478,Z 733.181,A -85,B 0,C 180,E1 -440.19,E2 -440.19} C_VEL
LIN {X 0,Y 608.485,Z 743.58,A -85,B 0,C 180,E1 -440.945,E2 -440.945} C_VEL
LIN {X 0,Y 608.475,Z 752.101,A -85,B 0,C 180,E1 -441.698,E2 -441.698} C_VEL
LIN {X 0,Y 608.471,Z 759.951,A -85,B 0,C 180,E1 -442.533,E2 -442.533} C_VEL
LIN {X 0,Y 608.462,Z 767.282,A -85,B 0,C 180,E1 -443.484,E2 -443.484} C_VEL
LIN {X 0,Y 608.45,Z 772.86,A -85,B 0,C 180,E1 -444.365,E2 -444.365} C_VEL
LIN {X 0,Y 608.432,Z 777.945,A -85,B 0,C 180,E1 -445.361,E2 -445.361} C_VEL
LIN {X 0,Y 608.449,Z 781.893,A -85,B 0,C 180,E1 -446.357,E2 -446.357} C_VEL
LIN {X 0,Y 608.425,Z 784.806,A -85,B 0,C 180,E1 -447.351,E2 -447.351} C_VEL
LIN {X 0,Y 608.443,Z 786.2,A -85,B 0,C 180,E1 -448.013,E2 -448.013} C_VEL
LIN {X 0,Y 608.438,Z 787.783,A -85,B 0,C 180,E1 -449.337,E2 -449.337} C_VEL
LIN {X 0,Y 608.434,Z 788,A -85,B 0,C 180,E1 -449.999,E2 -449.999} C_VEL
LIN {X 0,Y 608.448,Z 787.185,A -85,B 0,C 180,E1 -451.323,E2 -451.323} C_VEL
LIN {X 0,Y 608.443,Z 786.203,A -85,B 0,C 180,E1 -451.985,E2 -451.985} C_VEL
LIN {X 0,Y 608.425,Z 784.812,A -85,B 0,C 180,E1 -452.647,E2 -452.647} C_VEL
LIN {X 0,Y 608.449,Z 781.9,A -85,B 0,C 180,E1 -453.641,E2 -453.641} C_VEL
LIN {X 0,Y 608.432,Z 777.955,A -85,B 0,C 180,E1 -454.637,E2 -454.637} C_VEL
LIN {X 0,Y 608.437,Z 771.884,A -85,B 0,C 180,E1 -455.8,E2 -455.8} C_VEL
LIN {X 0,Y 608.461,Z 765.244,A -85,B 0,C 180,E1 -456.798,E2 -456.798} C_VEL
LIN {X 0,Y 608.455,Z 757,A -85,B 0,C 180,E1 -457.799,E2 -457.799} C_VEL
LIN {X 0,Y 608.472,Z 748.55,A -85,B 0,C 180,E1 -458.635,E2 -458.635} C_VEL
LIN {X 0,Y 608.477,Z 738.107,A -85,B 0,C 180,E1 -459.472,E2 -459.472} C_VEL
LIN {X 0,Y 608.488,Z 727.776,A -85,B 0,C 180,E1 -460.144,E2 -460.144} C_VEL
LIN {X 0,Y 608.522,Z 716.26,A -85,B 0,C 180,E1 -460.74,E2 -460.74} C_VEL
LIN {X 0,Y 608.533,Z 704.902,A -85,B 0,C 180,E1 -461.192,E2 -461.192} C_VEL
LIN {X 0,Y 608.555,Z 691.406,A -85,B 0,C 180,E1 -461.574,E2 -461.574} C_VEL
LIN {X 0,Y 608.547,Z 678.178,A -85,B 0,C 180,E1 -461.807,E2 -461.807} C_VEL
LIN {X 0,Y 608.529,Z 573.926,A -85,B 0,C 180,E1 -463.056,E2 -463.056} C_VEL
LIN {X 0,Y 608.509,Z 547.279,A -85,B 0,C 180,E1 -465.747,E2 -465.747} C_VEL
LIN {X 0,Y 608.554,Z 519.478,A -85,B 0,C 180,E1 -468.61,E2 -468.61} C_VEL
LIN {X 0,Y 608.631,Z 493.487,A -85,B 0,C 180,E1 -471.329,E2 -471.329} C_VEL
LIN {X 0,Y 608.706,Z 466.554,A -85,B 0,C 180,E1 -474.2,E2 -474.2} C_VEL
LIN {X 0,Y 608.703,Z 449.781,A -85,B 0,C 180,E1 -476.022,E2 -476.022} C_VEL
LIN {X 0,Y 608.48,Z 448.745,A -85,B 0,C 180,E1 -476.194,E2 -476.194} C_VEL
LIN {X 0,Y 608.4,Z 448.694,A -85,B 0,C 180,E1 -479.022,E2 -479.022} C_VEL
LIN {X 0,Y 608.422,Z 448.691,A -85,B 0,C 180,E1 -481.317,E2 -481.317} C_VEL
LIN {X 0,Y 608.44,Z 448.693,A -85,B 0,C 180,E1 -483.73,E2 -483.73} C_VEL
LIN {X 0,Y 608.436,Z 448.699,A -85,B 0,C 180,E1 -486.091,E2 -486.091} C_VEL
LIN {X 0,Y 608.415,Z 448.695,A -85,B 0,C 180,E1 -488.59,E2 -488.59} C_VEL
LIN {X 0,Y 608.412,Z 448.692,A -85,B 0,C 180,E1 -491.336,E2 -491.336} C_VEL
LIN {X 0,Y 608.451,Z 448.692,A -85,B 0,C 180,E1 -493.869,E2 -493.869} C_VEL
LIN {X 0,Y 608.457,Z 448.69,A -85,B 0,C 180,E1 -496.69,E2 -496.69} C_VEL
LIN {X 0,Y 608.432,Z 448.691,A -85,B 0,C 180,E1 -498.821,E2 -498.821} C_VEL
LIN {X 0,Y 608.439,Z 448.691,A -85,B 0,C 180,E1 -501.761,E2 -501.761} C_VEL
LIN {X 0,Y 608.433,Z 448.695,A -85,B 0,C 180,E1 -503.954,E2 -503.954} C_VEL
LIN {X 0,Y 608.461,Z 448.697,A -85,B 0,C 180,E1 -506.329,E2 -506.329} C_VEL
LIN {X 0,Y 608.465,Z 448.689,A -85,B 0,C 180,E1 -508.727,E2 -508.727} C_VEL
LIN {X 0,Y 608.43,Z 448.69,A -85,B 0,C 180,E1 -511.384,E2 -511.384} C_VEL
LIN {X 0,Y 608.425,Z 448.695,A -85,B 0,C 180,E1 -513.963,E2 -513.963} C_VEL
LIN {X 0,Y 608.433,Z 448.692,A -85,B 0,C 180,E1 -516.875,E2 -516.875} C_VEL
LIN {X 0,Y 608.43,Z 448.69,A -85,B 0,C 180,E1 -519.326,E2 -519.326} C_VEL
LIN {X 0,Y 608.414,Z 448.694,A -85,B 0,C 180,E1 -521.827,E2 -521.827} C_VEL
LIN {X 0,Y 608.47,Z 448.693,A -85,B 0,C 180,E1 -524.594,E2 -524.594} C_VEL
LIN {X 0,Y 608.447,Z 448.688,A -85,B 0,C 180,E1 -527.322,E2 -527.322} C_VEL
LIN {X 0,Y 608.433,Z 448.689,A -85,B 0,C 180,E1 -529.349,E2 -529.349} C_VEL
LIN {X 0,Y 608.453,Z 448.69,A -85,B 0,C 180,E1 -532.033,E2 -532.033} C_VEL
LIN {X 0,Y 608.469,Z 448.692,A -85,B 0,C 180,E1 -534.698,E2 -534.698} C_VEL
LIN {X 0,Y 608.451,Z 448.687,A -85,B 0,C 180,E1 -537.352,E2 -537.352} C_VEL
LIN {X 0,Y 608.445,Z 448.69,A -85,B 0,C 180,E1 -540,E2 -540} C_VEL
LIN {X 0,Y 608.485,Z 448.693,A -85,B 0,C 180,E1 -542.648,E2 -542.648} C_VEL
LIN {X 0,Y 608.453,Z 448.688,A -85,B 0,C 180,E1 -545.302,E2 -545.302} C_VEL
LIN {X 0,Y 608.45,Z 448.689,A -85,B 0,C 180,E1 -547.967,E2 -547.967} C_VEL
LIN {X 0,Y 608.445,Z 448.688,A -85,B 0,C 180,E1 -549.476,E2 -549.476} C_VEL
LIN {X 0,Y 607.754,Z 448.777,A -85,B 0,C 180,E1 -550.029,E2 -550.029} C_VEL
LIN {X 0,Y 604.89,Z 449.136,A -85,B 0,C 180,E1 -550.926,E2 -550.926} C_VEL
LIN {X 0,Y 602.493,Z 449.433,A -85,B 0,C 180,E1 -551.648,E2 -551.648} C_VEL
LIN {X 0,Y 601.475,Z 449.56,A -85,B 0,C 180,E1 -552.204,E2 -552.204} C_VEL
LIN {X 0,Y 601.396,Z 449.569,A -85,B 0,C 180,E1 -552.393,E2 -552.393} C_VEL
LIN {X 0,Y 601.426,Z 449.569,A -85,B 0,C 180,E1 -554.897,E2 -554.897} C_VEL
LIN {X 0,Y 601.385,Z 449.567,A -85,B 0,C 180,E1 -557.688,E2 -557.688} C_VEL
LIN {X 0,Y 601.423,Z 449.57,A -85,B 0,C 180,E1 -560.522,E2 -560.522} C_VEL
LIN {X 0,Y 601.409,Z 449.565,A -85,B 0,C 180,E1 -563.41,E2 -563.41} C_VEL
LIN {X 0,Y 601.392,Z 449.571,A -85,B 0,C 180,E1 -566.364,E2 -566.364} C_VEL
LIN {X 0,Y 601.434,Z 449.572,A -85,B 0,C 180,E1 -568.792,E2 -568.792} C_VEL
LIN {X 0,Y 601.4,Z 449.565,A -85,B 0,C 180,E1 -571.727,E2 -571.727} C_VEL
LIN {X 0,Y 601.419,Z 449.564,A -85,B 0,C 180,E1 -574.119,E2 -574.119} C_VEL
LIN {X 0,Y 601.399,Z 449.572,A -85,B 0,C 180,E1 -576.583,E2 -576.583} C_VEL
LIN {X 0,Y 601.43,Z 449.563,A -85,B 0,C 180,E1 -579.537,E2 -579.537} C_VEL
LIN {X 0,Y 601.413,Z 449.564,A -85,B 0,C 180,E1 -581.766,E2 -581.766} C_VEL
LIN {X 0,Y 601.413,Z 449.569,A -85,B 0,C 180,E1 -584.536,E2 -584.536} C_VEL
LIN {X 0,Y 601.431,Z 449.564,A -85,B 0,C 180,E1 -587.407,E2 -587.407} C_VEL
LIN {X 0,Y 601.403,Z 449.565,A -85,B 0,C 180,E1 -590.006,E2 -590.006} C_VEL
LIN {X 0,Y 601.43,Z 449.567,A -85,B 0,C 180,E1 -592.618,E2 -592.618} C_VEL
LIN {X 0,Y 601.431,Z 449.571,A -85,B 0,C 180,E1 -595.071,E2 -595.071} C_VEL
LIN {X 0,Y 601.436,Z 449.564,A -85,B 0,C 180,E1 -597.486,E2 -597.486} C_VEL
LIN {X 0,Y 601.42,Z 449.563,A -85,B 0,C 180,E1 -599.853,E2 -599.853} C_VEL
LIN {X 0,Y 601.416,Z 449.568,A -85,B 0,C 180,E1 -602.637,E2 -602.637} C_VEL
LIN {X 0,Y 601.402,Z 449.575,A -85,B 0,C 180,E1 -605.123,E2 -605.123} C_VEL
LIN {X 0,Y 601.411,Z 449.569,A -85,B 0,C 180,E1 -607.395,E2 -607.395} C_VEL
LIN {X 0,Y 601.403,Z 449.565,A -85,B 0,C 180,E1 -610.192,E2 -610.192} C_VEL
LIN {X 0,Y 601.429,Z 449.572,A -85,B 0,C 180,E1 -613.015,E2 -613.015} C_VEL
LIN {X 0,Y 601.418,Z 449.564,A -85,B 0,C 180,E1 -615.909,E2 -615.909} C_VEL
LIN {X 0,Y 601.433,Z 449.563,A -85,B 0,C 180,E1 -618.543,E2 -618.543} C_VEL
LIN {X 0,Y 601.435,Z 449.57,A -85,B 0,C 180,E1 -621.264,E2 -621.264} C_VEL
LIN {X 0,Y 601.433,Z 449.562,A -85,B 0,C 180,E1 -623.964,E2 -623.964} C_VEL
LIN {X 0,Y 601.427,Z 449.565,A -85,B 0,C 180,E1 -626.652,E2 -626.652} C_VEL
LIN {X 0,Y 601.456,Z 449.568,A -85,B 0,C 180,E1 -629.332,E2 -629.332} C_VEL
LIN {X 0,Y 601.451,Z 449.716,A -85,B 0,C 180,E1 -631.047,E2 -631.047} C_VEL
LIN {X 0,Y 601.609,Z 450.511,A -85,B 0,C 180,E1 -631.152,E2 -631.152} C_VEL
LIN {X 0,Y 601.646,Z 485.564,A -85,B 0,C 180,E1 -631.591,E2 -631.591} C_VEL
LIN {X 0,Y 601.629,Z 534.639,A -85,B 0,C 180,E1 -632.198,E2 -632.198} C_VEL
LIN {X 0,Y 601.571,Z 548.261,A -85,B 0,C 180,E1 -632.512,E2 -632.512} C_VEL
LIN {X 0,Y 601.573,Z 560.484,A -85,B 0,C 180,E1 -632.931,E2 -632.931} C_VEL
LIN {X 0,Y 601.519,Z 571.498,A -85,B 0,C 180,E1 -633.434,E2 -633.434} C_VEL
LIN {X 0,Y 601.503,Z 582.958,A -85,B 0,C 180,E1 -634.105,E2 -634.105} C_VEL
LIN {X 0,Y 601.443,Z 593.308,A -85,B 0,C 180,E1 -634.861,E2 -634.861} C_VEL
LIN {X 0,Y 601.428,Z 602.688,A -85,B 0,C 180,E1 -635.701,E2 -635.701} C_VEL
LIN {X 0,Y 601.407,Z 611.754,A -85,B 0,C 180,E1 -636.712,E2 -636.712} C_VEL
LIN {X 0,Y 601.386,Z 619.096,A -85,B 0,C 180,E1 -637.725,E2 -637.725} C_VEL
LIN {X 0,Y 601.381,Z 624.998,A -85,B 0,C 180,E1 -638.739,E2 -638.739} C_VEL
LIN {X 0,Y 601.341,Z 629.665,A -85,B 0,C 180,E1 -639.758,E2 -639.758} C_VEL
LIN {X 0,Y 601.352,Z 633.786,A -85,B 0,C 180,E1 -640.977,E2 -640.977} C_VEL
LIN {X 0,Y 601.342,Z 636.382,A -85,B 0,C 180,E1 -642.145,E2 -642.145} C_VEL
LIN {X 0,Y 601.324,Z 637.331,A -85,B 0,C 180,E1 -642.831,E2 -642.831} C_VEL
LIN {X 0,Y 601.349,Z 637.999,A -85,B 0,C 180,E1 -644.065,E2 -644.065} C_VEL
LIN {X 0,Y 601.315,Z 637.654,A -85,B 0,C 180,E1 -644.901,E2 -644.901} C_VEL
LIN {X 0,Y 601.324,Z 636.937,A -85,B 0,C 180,E1 -645.595,E2 -645.595} C_VEL
LIN {X 0,Y 601.322,Z 635.113,A -85,B 0,C 180,E1 -646.589,E2 -646.589} C_VEL
LIN {X 0,Y 601.326,Z 632.021,A -85,B 0,C 180,E1 -647.691,E2 -647.691} C_VEL
LIN {X 0,Y 601.35,Z 627.672,A -85,B 0,C 180,E1 -648.801,E2 -648.801} C_VEL
LIN {X 0,Y 601.369,Z 621.424,A -85,B 0,C 180,E1 -649.99,E2 -649.99} C_VEL
LIN {X 0,Y 601.375,Z 613.98,A -85,B 0,C 180,E1 -651.096,E2 -651.096} C_VEL
LIN {X 0,Y 601.386,Z 606.78,A -85,B 0,C 180,E1 -651.961,E2 -651.961} C_VEL
LIN {X 0,Y 601.42,Z 597.596,A -85,B 0,C 180,E1 -652.865,E2 -652.865} C_VEL
LIN {X 0,Y 601.459,Z 587.361,A -85,B 0,C 180,E1 -653.684,E2 -653.684} C_VEL
LIN {X 0,Y 601.495,Z 576.064,A -85,B 0,C 180,E1 -654.409,E2 -654.409} C_VEL
LIN {X 0,Y 601.537,Z 563.958,A -85,B 0,C 180,E1 -655.012,E2 -655.012} C_VEL
LIN {X 0,Y 601.556,Z 551.704,A -85,B 0,C 180,E1 -655.474,E2 -655.474} C_VEL
LIN {X 0,Y 601.621,Z 538.854,A -85,B 0,C 180,E1 -655.813,E2 -655.813} C_VEL
LIN {X 0,Y 601.635,Z 524.041,A -85,B 0,C 180,E1 -656.039,E2 -656.039} C_VEL
LIN {X 0,Y 601.68,Z 450.752,A -85,B 0,C 180,E1 -656.925,E2 -656.925} C_VEL
LIN {X 0,Y 601.449,Z 449.696,A -85,B 0,C 180,E1 -657.042,E2 -657.042} C_VEL
LIN {X 0,Y 601.412,Z 449.568,A -85,B 0,C 180,E1 -659.395,E2 -659.395} C_VEL
LIN {X 0,Y 601.404,Z 449.566,A -85,B 0,C 180,E1 -661.728,E2 -661.728} C_VEL
LIN {X 0,Y 601.423,Z 449.564,A -85,B 0,C 180,E1 -664.12,E2 -664.12} C_VEL
LIN {X 0,Y 601.439,Z 449.563,A -85,B 0,C 180,E1 -667.383,E2 -667.383} C_VEL
LIN {X 0,Y 601.404,Z 449.565,A -85,B 0,C 180,E1 -669.997,E2 -669.997} C_VEL
LIN {X 0,Y 601.415,Z 449.572,A -85,B 0,C 180,E1 -672.671,E2 -672.671} C_VEL
LIN {X 0,Y 601.402,Z 449.567,A -85,B 0,C 180,E1 -675.48,E2 -675.48} C_VEL
LIN {X 0,Y 601.425,Z 449.567,A -85,B 0,C 180,E1 -678.408,E2 -678.408} C_VEL
LIN {X 0,Y 601.407,Z 449.575,A -85,B 0,C 180,E1 -680.873,E2 -680.873} C_VEL
LIN {X 0,Y 601.404,Z 449.57,A -85,B 0,C 180,E1 -683.417,E2 -683.417} C_VEL
LIN {X 0,Y 601.454,Z 449.723,A -85,B 0,C 180,E1 -684.635,E2 -684.635} C_VEL
LIN {X 0,Y 601.653,Z 454.058,A -85,B 0,C 180,E1 -685.288,E2 -685.288} C_VEL
LIN {X 0,Y 601.558,Z 473.899,A -85,B 0,C 180,E1 -688.086,E2 -688.086} C_VEL
LIN {X 0,Y 601.52,Z 493.302,A -85,B 0,C 180,E1 -690.779,E2 -690.779} C_VEL
LIN {X 0,Y 601.455,Z 514.196,A -85,B 0,C 180,E1 -693.639,E2 -693.639} C_VEL
LIN {X 0,Y 601.471,Z 516.085,A -85,B 0,C 180,E1 -693.857,E2 -693.857} C_VEL
LIN {X 0,Y 601.68,Z 520.837,A -85,B 0,C 180,E1 -693.935,E2 -693.935} C_VEL
LIN {X 0,Y 601.588,Z 624.615,A -85,B 0,C 180,E1 -695.196,E2 -695.196} C_VEL
LIN {X 0,Y 601.588,Z 638.514,A -85,B 0,C 180,E1 -695.519,E2 -695.519} C_VEL
LIN {X 0,Y 601.552,Z 651.084,A -85,B 0,C 180,E1 -695.956,E2 -695.956} C_VEL
LIN {X 0,Y 601.514,Z 662.781,A -85,B 0,C 180,E1 -696.503,E2 -696.503} C_VEL
LIN {X 0,Y 601.468,Z 674.826,A -85,B 0,C 180,E1 -697.229,E2 -697.229} C_VEL
LIN {X 0,Y 601.433,Z 685.503,A -85,B 0,C 180,E1 -698.042,E2 -698.042} C_VEL
LIN {X 0,Y 601.436,Z 694.665,A -85,B 0,C 180,E1 -698.906,E2 -698.906} C_VEL
LIN {X 0,Y 601.392,Z 702.737,A -85,B 0,C 180,E1 -699.834,E2 -699.834} C_VEL
LIN {X 0,Y 601.368,Z 710.222,A -85,B 0,C 180,E1 -700.9,E2 -700.9} C_VEL
LIN {X 0,Y 601.36,Z 716.088,A -85,B 0,C 180,E1 -701.959,E2 -701.959} C_VEL
LIN {X 0,Y 601.366,Z 720.63,A -85,B 0,C 180,E1 -703.012,E2 -703.012} C_VEL
LIN {X 0,Y 601.35,Z 723.008,A -85,B 0,C 180,E1 -703.711,E2 -703.711} C_VEL
LIN {X 0,Y 601.328,Z 724.908,A -85,B 0,C 180,E1 -704.407,E2 -704.407} C_VEL
LIN {X 0,Y 601.316,Z 726.31,A -85,B 0,C 180,E1 -705.1,E2 -705.1} C_VEL
LIN {X 0,Y 601.354,Z 727.449,A -85,B 0,C 180,E1 -705.937,E2 -705.937} C_VEL
LIN {X 0,Y 601.324,Z 727.977,A -85,B 0,C 180,E1 -707.17,E2 -707.17} C_VEL
LIN {X 0,Y 601.342,Z 727.687,A -85,B 0,C 180,E1 -707.856,E2 -707.856} C_VEL
LIN {X 0,Y 601.353,Z 726.248,A -85,B 0,C 180,E1 -709.027,E2 -709.027} C_VEL
LIN {X 0,Y 601.328,Z 724.339,A -85,B 0,C 180,E1 -709.903,E2 -709.903} C_VEL
LIN {X 0,Y 601.349,Z 721.201,A -85,B 0,C 180,E1 -710.922,E2 -710.922} C_VEL
LIN {X 0,Y 601.35,Z 717.014,A -85,B 0,C 180,E1 -711.938,E2 -711.938} C_VEL
LIN {X 0,Y 601.384,Z 710.64,A -85,B 0,C 180,E1 -713.121,E2 -713.121} C_VEL
LIN {X 0,Y 601.386,Z 703.718,A -85,B 0,C 180,E1 -714.131,E2 -714.131} C_VEL
LIN {X 0,Y 601.404,Z 695.091,A -85,B 0,C 180,E1 -715.14,E2 -715.14} C_VEL
LIN {X 0,Y 601.422,Z 686.288,A -85,B 0,C 180,E1 -715.98,E2 -715.98} C_VEL
LIN {X 0,Y 601.483,Z 675.452,A -85,B 0,C 180,E1 -716.819,E2 -716.819} C_VEL
LIN {X 0,Y 601.508,Z 664.594,A -85,B 0,C 180,E1 -717.489,E2 -717.489} C_VEL
LIN {X 0,Y 601.529,Z 652.5,A -85,B 0,C 180,E1 -718.075,E2 -718.075} C_VEL
LIN {X 0,Y 601.604,Z 639.721,A -85,B 0,C 180,E1 -718.536,E2 -718.536} C_VEL
LIN {X 0,Y 601.61,Z 626.944,A -85,B 0,C 180,E1 -718.85,E2 -718.85} C_VEL
LIN {X 0,Y 601.641,Z 608.859,A -85,B 0,C 180,E1 -719.101,E2 -719.101} C_VEL
LIN {X 0,Y 601.541,Z 516.805,A -85,B 0,C 180,E1 -720.209,E2 -720.209} C_VEL
LIN {X 0,Y 601.425,Z 515.427,A -85,B 0,C 180,E1 -720.293,E2 -720.293} C_VEL
LIN {X 0,Y 601.517,Z 495.564,A -85,B 0,C 180,E1 -723.014,E2 -723.014} C_VEL
LIN {X 0,Y 601.573,Z 475.064,A -85,B 0,C 180,E1 -725.867,E2 -725.867} C_VEL
LIN {X 0,Y 601.664,Z 454.8,A -85,B 0,C 180,E1 -728.735,E2 -728.735} C_VEL
LIN {X 0,Y 601.454,Z 449.686,A -85,B 0,C 180,E1 -729.5,E2 -729.5} C_VEL
LIN {X 0,Y 601.394,Z 449.568,A -85,B 0,C 180,E1 -732.143,E2 -732.143} C_VEL
LIN {X 0,Y 601.397,Z 449.573,A -85,B 0,C 180,E1 -734.898,E2 -734.898} C_VEL
LIN {X 0,Y 601.387,Z 449.57,A -85,B 0,C 180,E1 -737.689,E2 -737.689} C_VEL
LIN {X 0,Y 601.394,Z 449.568,A -85,B 0,C 180,E1 -739.81,E2 -739.81} C_VEL
LIN {X 0,Y 601.409,Z 449.571,A -85,B 0,C 180,E1 -742.683,E2 -742.683} C_VEL
LIN {X 0,Y 601.441,Z 449.562,A -85,B 0,C 180,E1 -745.617,E2 -745.617} C_VEL
LIN {X 0,Y 601.401,Z 449.566,A -85,B 0,C 180,E1 -747.869,E2 -747.869} C_VEL
LIN {X 0,Y 601.412,Z 449.566,A -85,B 0,C 180,E1 -750.165,E2 -750.165} C_VEL
LIN {X 0,Y 601.422,Z 449.574,A -85,B 0,C 180,E1 -752.714,E2 -752.714} C_VEL
LIN {X 0,Y 601.407,Z 449.569,A -85,B 0,C 180,E1 -755.112,E2 -755.112} C_VEL
LIN {X 0,Y 601.441,Z 449.561,A -85,B 0,C 180,E1 -757.419,E2 -757.419} C_VEL
LIN {X 0,Y 601.41,Z 449.567,A -85,B 0,C 180,E1 -759.995,E2 -759.995} C_VEL
LIN {X 0,Y 601.413,Z 449.572,A -85,B 0,C 180,E1 -762.67,E2 -762.67} C_VEL
LIN {X 0,Y 601.406,Z 449.566,A -85,B 0,C 180,E1 -765.479,E2 -765.479} C_VEL
LIN {X 0,Y 601.424,Z 449.573,A -85,B 0,C 180,E1 -768.407,E2 -768.407} C_VEL
LIN {X 0,Y 601.401,Z 449.567,A -85,B 0,C 180,E1 -770.872,E2 -770.872} C_VEL
LIN {X 0,Y 601.394,Z 449.567,A -85,B 0,C 180,E1 -773.415,E2 -773.415} C_VEL
LIN {X 0,Y 601.421,Z 449.572,A -85,B 0,C 180,E1 -776.066,E2 -776.066} C_VEL
LIN {X 0,Y 601.417,Z 449.568,A -85,B 0,C 180,E1 -778.546,E2 -778.546} C_VEL
LIN {X 0,Y 601.417,Z 449.566,A -85,B 0,C 180,E1 -781.371,E2 -781.371} C_VEL
LIN {X 0,Y 601.455,Z 449.806,A -85,B 0,C 180,E1 -783.689,E2 -783.689} C_VEL
LIN {X 0,Y 601.994,Z 452.462,A -85,B 0,C 180,E1 -784.019,E2 -784.019} C_VEL
LIN {X 0,Y 601.816,Z 478.096,A -85,B 0,C 180,E1 -786.805,E2 -786.805} C_VEL
LIN {X 0,Y 601.741,Z 503.243,A -85,B 0,C 180,E1 -789.488,E2 -789.488} C_VEL
LIN {X 0,Y 601.602,Z 530.247,A -85,B 0,C 180,E1 -792.317,E2 -792.317} C_VEL
LIN {X 0,Y 601.512,Z 553.875,A -85,B 0,C 180,E1 -794.758,E2 -794.758} C_VEL
LIN {X 0,Y 601.518,Z 573.858,A -85,B 0,C 180,E1 -796.786,E2 -796.786} C_VEL
LIN {X 0,Y 601.679,Z 577.845,A -85,B 0,C 180,E1 -796.854,E2 -796.854} C_VEL
LIN {X 0,Y 601.61,Z 683.891,A -85,B 0,C 180,E1 -798.138,E2 -798.138} C_VEL
LIN {X 0,Y 601.59,Z 697.18,A -85,B 0,C 180,E1 -798.437,E2 -798.437} C_VEL
LIN {X 0,Y 601.551,Z 708.904,A -85,B 0,C 180,E1 -798.825,E2 -798.825} C_VEL
LIN {X 0,Y 601.53,Z 719.901,A -85,B 0,C 180,E1 -799.31,E2 -799.31} C_VEL
LIN {X 0,Y 601.472,Z 730.563,A -85,B 0,C 180,E1 -799.905,E2 -799.905} C_VEL
LIN {X 0,Y 601.448,Z 741.462,A -85,B 0,C 180,E1 -800.668,E2 -800.668} C_VEL
LIN {X 0,Y 601.429,Z 752.101,A -85,B 0,C 180,E1 -801.6,E2 -801.6} C_VEL
LIN {X 0,Y 601.418,Z 759.951,A -85,B 0,C 180,E1 -802.445,E2 -802.445} C_VEL
LIN {X 0,Y 601.371,Z 767.219,A -85,B 0,C 180,E1 -803.397,E2 -803.397} C_VEL
LIN {X 0,Y 601.372,Z 772.86,A -85,B 0,C 180,E1 -804.298,E2 -804.298} C_VEL
LIN {X 0,Y 601.336,Z 777.945,A -85,B 0,C 180,E1 -805.306,E2 -805.306} C_VEL
LIN {X 0,Y 601.368,Z 781.892,A -85,B 0,C 180,E1 -806.314,E2 -806.314} C_VEL
LIN {X 0,Y 601.325,Z 784.806,A -85,B 0,C 180,E1 -807.319,E2 -807.319} C_VEL
LIN {X 0,Y 601.342,Z 786.2,A -85,B 0,C 180,E1 -807.99,E2 -807.99} C_VEL
LIN {X 0,Y 601.339,Z 787.783,A -85,B 0,C 180,E1 -809.329,E2 -809.329} C_VEL
LIN {X 0,Y 601.335,Z 788,A -85,B 0,C 180,E1 -809.999,E2 -809.999} C_VEL
LIN {X 0,Y 601.347,Z 787.186,A -85,B 0,C 180,E1 -811.338,E2 -811.338} C_VEL
LIN {X 0,Y 601.342,Z 786.204,A -85,B 0,C 180,E1 -812.008,E2 -812.008} C_VEL
LIN {X 0,Y 601.325,Z 784.812,A -85,B 0,C 180,E1 -812.678,E2 -812.678} C_VEL
LIN {X 0,Y 601.368,Z 781.9,A -85,B 0,C 180,E1 -813.684,E2 -813.684} C_VEL
LIN {X 0,Y 601.336,Z 777.955,A -85,B 0,C 180,E1 -814.692,E2 -814.692} C_VEL
LIN {X 0,Y 601.372,Z 771.884,A -85,B 0,C 180,E1 -815.868,E2 -815.868} C_VEL
LIN {X 0,Y 601.387,Z 765.244,A -85,B 0,C 180,E1 -816.878,E2 -816.878} C_VEL
LIN {X 0,Y 601.4,Z 757,A -85,B 0,C 180,E1 -817.891,E2 -817.891} C_VEL
LIN {X 0,Y 601.436,Z 748.55,A -85,B 0,C 180,E1 -818.736,E2 -818.736} C_VEL
LIN {X 0,Y 601.445,Z 738.109,A -85,B 0,C 180,E1 -819.584,E2 -819.584} C_VEL
LIN {X 0,Y 601.484,Z 727.777,A -85,B 0,C 180,E1 -820.263,E2 -820.263} C_VEL
LIN {X 0,Y 601.538,Z 716.914,A -85,B 0,C 180,E1 -820.835,E2 -820.835} C_VEL
LIN {X 0,Y 601.564,Z 704.406,A -85,B 0,C 180,E1 -821.339,E2 -821.339} C_VEL
LIN {X 0,Y 601.6,Z 691.405,A -85,B 0,C 180,E1 -821.71,E2 -821.71} C_VEL
LIN {X 0,Y 601.614,Z 678.178,A -85,B 0,C 180,E1 -821.945,E2 -821.945} C_VEL
LIN {X 0,Y 601.576,Z 574.615,A -85,B 0,C 180,E1 -823.188,E2 -823.188} C_VEL
LIN {X 0,Y 601.518,Z 573.359,A -85,B 0,C 180,E1 -823.254,E2 -823.254} C_VEL
LIN {X 0,Y 601.564,Z 545.598,A -85,B 0,C 180,E1 -826.108,E2 -826.108} C_VEL
LIN {X 0,Y 601.646,Z 518.998,A -85,B 0,C 180,E1 -828.882,E2 -828.882} C_VEL
LIN {X 0,Y 601.762,Z 493.487,A -85,B 0,C 180,E1 -831.584,E2 -831.584} C_VEL
LIN {X 0,Y 601.891,Z 467.503,A -85,B 0,C 180,E1 -834.388,E2 -834.388} C_VEL
LIN {X 0,Y 601.962,Z 452.006,A -85,B 0,C 180,E1 -836.089,E2 -836.089} C_VEL
LIN {X 0,Y 601.419,Z 449.637,A -85,B 0,C 180,E1 -836.42,E2 -836.42} C_VEL
LIN {X 0,Y 601.376,Z 449.57,A -85,B 0,C 180,E1 -839.394,E2 -839.394} C_VEL
LIN {X 0,Y 601.39,Z 449.572,A -85,B 0,C 180,E1 -841.726,E2 -841.726} C_VEL
LIN {X 0,Y 601.409,Z 449.576,A -85,B 0,C 180,E1 -844.118,E2 -844.118} C_VEL
LIN {X 0,Y 601.376,Z 449.572,A -85,B 0,C 180,E1 -846.583,E2 -846.583} C_VEL
LIN {X 0,Y 601.374,Z 449.569,A -85,B 0,C 180,E1 -849.128,E2 -849.128} C_VEL
LIN {X 0,Y 601.407,Z 449.568,A -85,B 0,C 180,E1 -851.765,E2 -851.765} C_VEL
LIN {X 0,Y 601.388,Z 449.572,A -85,B 0,C 180,E1 -854.531,E2 -854.531} C_VEL
LIN {X 0,Y 601.419,Z 449.57,A -85,B 0,C 180,E1 -856.426,E2 -856.426} C_VEL
LIN {X 0,Y 601.394,Z 449.566,A -85,B 0,C 180,E1 -859.124,E2 -859.124} C_VEL
LIN {X 0,Y 601.39,Z 449.569,A -85,B 0,C 180,E1 -861.729,E2 -861.729} C_VEL
LIN {X 0,Y 601.376,Z 449.579,A -85,B 0,C 180,E1 -864.244,E2 -864.244} C_VEL
LIN {X 0,Y 601.415,Z 449.568,A -85,B 0,C 180,E1 -866.685,E2 -866.685} C_VEL
LIN {X 0,Y 601.402,Z 449.566,A -85,B 0,C 180,E1 -869.057,E2 -869.057} C_VEL
LIN {X 0,Y 601.39,Z 449.567,A -85,B 0,C 180,E1 -871.371,E2 -871.371} C_VEL
LIN {X 0,Y 601.378,Z 449.569,A -85,B 0,C 180,E1 -873.635,E2 -873.635} C_VEL
LIN {X 0,Y 601.403,Z 449.572,A -85,B 0,C 180,E1 -876.589,E2 -876.589} C_VEL
LIN {X 0,Y 601.395,Z 449.566,A -85,B 0,C 180,E1 -879.477,E2 -879.477} C_VEL
LIN {X 0,Y 601.384,Z 449.577,A -85,B 0,C 180,E1 -882.311,E2 -882.311} C_VEL
LIN {X 0,Y 601.393,Z 449.567,A -85,B 0,C 180,E1 -885.102,E2 -885.102} C_VEL
LIN {X 0,Y 601.394,Z 449.568,A -85,B 0,C 180,E1 -887.857,E2 -887.857} C_VEL
LIN {X 0,Y 601.407,Z 449.567,A -85,B 0,C 180,E1 -889.904,E2 -889.904} C_VEL
LIN {X 0,Y 601.447,Z 449.568,A -85,B 0,C 180,E1 -892.615,E2 -892.615} C_VEL
LIN {X 0,Y 601.397,Z 449.566,A -85,B 0,C 180,E1 -895.308,E2 -895.308} C_VEL
LIN {X 0,Y 601.419,Z 449.563,A -85,B 0,C 180,E1 -897.321,E2 -897.321} C_VEL
LIN {X 0,Y 601.415,Z 449.566,A -85,B 0,C 180,E1 -900,E2 -900} C_VEL
LIN {X 0,Y 601.448,Z 449.569,A -85,B 0,C 180,E1 -902.679,E2 -902.679} C_VEL
LIN {X 0,Y 601.414,Z 449.564,A -85,B 0,C 180,E1 -905.364,E2 -905.364} C_VEL
LIN {X 0,Y 601.419,Z 449.565,A -85,B 0,C 180,E1 -908.061,E2 -908.061} C_VEL
LIN {X 0,Y 601.424,Z 449.567,A -85,B 0,C 180,E1 -911.02,E2 -911.02} C_VEL
LIN {X 0,Y 601.396,Z 449.569,A -85,B 0,C 180,E1 -912.393,E2 -912.393} C_VEL
LIN {X 0,Y 600.744,Z 449.655,A -85,B 0,C 180,E1 -912.952,E2 -912.952} C_VEL
LIN {X 0,Y 597.898,Z 450.009,A -85,B 0,C 180,E1 -913.86,E2 -913.86} C_VEL
LIN {X 0,Y 595.481,Z 450.313,A -85,B 0,C 180,E1 -914.59,E2 -914.59} C_VEL
LIN {X 0,Y 594.439,Z 450.436,A -85,B 0,C 180,E1 -915.154,E2 -915.154} C_VEL
LIN {X 0,Y 594.351,Z 450.445,A -85,B 0,C 180,E1 -915.345,E2 -915.345} C_VEL
LIN {X 0,Y 594.342,Z 450.445,A -85,B 0,C 180,E1 -917.905,E2 -917.905} C_VEL
LIN {X 0,Y 594.399,Z 450.447,A -85,B 0,C 180,E1 -920.775,E2 -920.775} C_VEL
LIN {X 0,Y 594.374,Z 450.441,A -85,B 0,C 180,E1 -923.704,E2 -923.704} C_VEL
LIN {X 0,Y 594.378,Z 450.451,A -85,B 0,C 180,E1 -926.7,E2 -926.7} C_VEL
LIN {X 0,Y 594.373,Z 450.447,A -85,B 0,C 180,E1 -928.999,E2 -928.999} C_VEL
LIN {X 0,Y 594.379,Z 450.44,A -85,B 0,C 180,E1 -931.646,E2 -931.646} C_VEL
LIN {X 0,Y 594.391,Z 450.445,A -85,B 0,C 180,E1 -934.579,E2 -934.579} C_VEL
LIN {X 0,Y 594.379,Z 450.441,A -85,B 0,C 180,E1 -937.61,E2 -937.61} C_VEL
LIN {X 0,Y 594.361,Z 450.448,A -85,B 0,C 180,E1 -940.567,E2 -940.567} C_VEL
LIN {X 0,Y 594.368,Z 450.445,A -85,B 0,C 180,E1 -943.299,E2 -943.299} C_VEL
LIN {X 0,Y 594.371,Z 450.442,A -85,B 0,C 180,E1 -946.16,E2 -946.16} C_VEL
LIN {X 0,Y 594.375,Z 450.445,A -85,B 0,C 180,E1 -948.538,E2 -948.538} C_VEL
LIN {X 0,Y 594.38,Z 450.444,A -85,B 0,C 180,E1 -951.296,E2 -951.296} C_VEL
LIN {X 0,Y 594.377,Z 450.441,A -85,B 0,C 180,E1 -953.759,E2 -953.759} C_VEL
LIN {X 0,Y 594.369,Z 450.442,A -85,B 0,C 180,E1 -956.24,E2 -956.24} C_VEL
LIN {X 0,Y 594.385,Z 450.444,A -85,B 0,C 180,E1 -958.652,E2 -958.652} C_VEL
LIN {X 0,Y 594.379,Z 450.45,A -85,B 0,C 180,E1 -961.042,E2 -961.042} C_VEL
LIN {X 0,Y 594.378,Z 450.44,A -85,B 0,C 180,E1 -963.978,E2 -963.978} C_VEL
LIN {X 0,Y 594.384,Z 450.44,A -85,B 0,C 180,E1 -966.297,E2 -966.297} C_VEL
LIN {X 0,Y 594.403,Z 450.445,A -85,B 0,C 180,E1 -969.226,E2 -969.226} C_VEL
LIN {X 0,Y 594.35,Z 450.444,A -85,B 0,C 180,E1 -972.096,E2 -972.096} C_VEL
LIN {X 0,Y 594.366,Z 450.442,A -85,B 0,C 180,E1 -974.22,E2 -974.22} C_VEL
LIN {X 0,Y 594.368,Z 450.451,A -85,B 0,C 180,E1 -977.018,E2 -977.018} C_VEL
LIN {X 0,Y 594.39,Z 450.44,A -85,B 0,C 180,E1 -979.785,E2 -979.785} C_VEL
LIN {X 0,Y 594.393,Z 450.44,A -85,B 0,C 180,E1 -982.528,E2 -982.528} C_VEL
LIN {X 0,Y 594.393,Z 450.449,A -85,B 0,C 180,E1 -985.254,E2 -985.254} C_VEL
LIN {X 0,Y 594.403,Z 450.439,A -85,B 0,C 180,E1 -987.968,E2 -987.968} C_VEL
LIN {X 0,Y 594.416,Z 450.442,A -85,B 0,C 180,E1 -990.679,E2 -990.679} C_VEL
LIN {X 0,Y 594.443,Z 450.714,A -85,B 0,C 180,E1 -990.933,E2 -990.933} C_VEL
LIN {X 0,Y 594.676,Z 451.846,A -85,B 0,C 180,E1 -991.027,E2 -991.027} C_VEL
LIN {X 0,Y 594.695,Z 534.449,A -85,B 0,C 180,E1 -992.054,E2 -992.054} C_VEL
LIN {X 0,Y 594.604,Z 548.158,A -85,B 0,C 180,E1 -992.372,E2 -992.372} C_VEL
LIN {X 0,Y 594.59,Z 560.414,A -85,B 0,C 180,E1 -992.796,E2 -992.796} C_VEL
LIN {X 0,Y 594.518,Z 571.446,A -85,B 0,C 180,E1 -993.305,E2 -993.305} C_VEL
LIN {X 0,Y 594.475,Z 582.925,A -85,B 0,C 180,E1 -993.984,E2 -993.984} C_VEL
LIN {X 0,Y 594.419,Z 593.275,A -85,B 0,C 180,E1 -994.749,E2 -994.749} C_VEL
LIN {X 0,Y 594.392,Z 602.658,A -85,B 0,C 180,E1 -995.599,E2 -995.599} C_VEL
LIN {X 0,Y 594.336,Z 611.882,A -85,B 0,C 180,E1 -996.64,E2 -996.64} C_VEL
LIN {X 0,Y 594.299,Z 619.079,A -85,B 0,C 180,E1 -997.646,E2 -997.646} C_VEL
LIN {X 0,Y 594.292,Z 625.834,A -85,B 0,C 180,E1 -998.845,E2 -998.845} C_VEL
LIN {X 0,Y 594.257,Z 630.31,A -85,B 0,C 180,E1 -999.875,E2 -999.875} C_VEL
LIN {X 0,Y 594.262,Z 633.973,A -85,B 0,C 180,E1 -1001.011,E2 -1001.011} C_VEL
LIN {X 0,Y 594.239,Z 636.659,A -85,B 0,C 180,E1 -1002.292,E2 -1002.292} C_VEL
LIN {X 0,Y 594.243,Z 637.517,A -85,B 0,C 180,E1 -1002.987,E2 -1002.987} C_VEL
LIN {X 0,Y 594.26,Z 637.988,A -85,B 0,C 180,E1 -1004.125,E2 -1004.125} C_VEL
LIN {X 0,Y 594.209,Z 637.533,A -85,B 0,C 180,E1 -1005.083,E2 -1005.083} C_VEL
LIN {X 0,Y 594.222,Z 636.676,A -85,B 0,C 180,E1 -1005.786,E2 -1005.786} C_VEL
LIN {X 0,Y 594.238,Z 635.005,A -85,B 0,C 180,E1 -1006.669,E2 -1006.669} C_VEL
LIN {X 0,Y 594.241,Z 631.422,A -85,B 0,C 180,E1 -1007.91,E2 -1007.91} C_VEL
LIN {X 0,Y 594.28,Z 626.625,A -85,B 0,C 180,E1 -1009.079,E2 -1009.079} C_VEL
LIN {X 0,Y 594.298,Z 620.374,A -85,B 0,C 180,E1 -1010.238,E2 -1010.238} C_VEL
LIN {X 0,Y 594.343,Z 612.79,A -85,B 0,C 180,E1 -1011.335,E2 -1011.335} C_VEL
LIN {X 0,Y 594.372,Z 603.725,A -85,B 0,C 180,E1 -1012.38,E2 -1012.38} C_VEL
LIN {X 0,Y 594.418,Z 594.496,A -85,B 0,C 180,E1 -1013.242,E2 -1013.242} C_VEL
LIN {X 0,Y 594.441,Z 583.422,A -85,B 0,C 180,E1 -1014.073,E2 -1014.073} C_VEL
LIN {X 0,Y 594.541,Z 571.614,A -85,B 0,C 180,E1 -1014.776,E2 -1014.776} C_VEL
LIN {X 0,Y 594.575,Z 559.61,A -85,B 0,C 180,E1 -1015.325,E2 -1015.325} C_VEL
LIN {X 0,Y 594.64,Z 546.367,A -85,B 0,C 180,E1 -1015.768,E2 -1015.768} C_VEL
LIN {X 0,Y 594.674,Z 533.228,A -85,B 0,C 180,E1 -1016.058,E2 -1016.058} C_VEL
LIN {X 0,Y 594.636,Z 451.671,A -85,B 0,C 180,E1 -1017.068,E2 -1017.068} C_VEL
LIN {X 0,Y 594.427,Z 450.624,A -85,B 0,C 180,E1 -1017.173,E2 -1017.173} C_VEL
LIN {X 0,Y 594.376,Z 450.442,A -85,B 0,C 180,E1 -1019.777,E2 -1019.777} C_VEL
LIN {X 0,Y 594.371,Z 450.443,A -85,B 0,C 180,E1 -1022.148,E2 -1022.148} C_VEL
LIN {X 0,Y 594.383,Z 450.446,A -85,B 0,C 180,E1 -1024.581,E2 -1024.581} C_VEL
LIN {X 0,Y 594.391,Z 450.44,A -85,B 0,C 180,E1 -1027.609,E2 -1027.609} C_VEL
LIN {X 0,Y 594.37,Z 450.447,A -85,B 0,C 180,E1 -1030.568,E2 -1030.568} C_VEL
LIN {X 0,Y 594.371,Z 450.445,A -85,B 0,C 180,E1 -1033.3,E2 -1033.3} C_VEL
LIN {X 0,Y 594.364,Z 450.444,A -85,B 0,C 180,E1 -1036.162,E2 -1036.162} C_VEL
LIN {X 0,Y 594.383,Z 450.446,A -85,B 0,C 180,E1 -1038.537,E2 -1038.537} C_VEL
LIN {X 0,Y 594.373,Z 450.445,A -85,B 0,C 180,E1 -1041.298,E2 -1041.298} C_VEL
LIN {X 0,Y 594.374,Z 450.447,A -85,B 0,C 180,E1 -1044.176,E2 -1044.176} C_VEL
LIN {X 0,Y 594.43,Z 450.636,A -85,B 0,C 180,E1 -1044.493,E2 -1044.493} C_VEL
LIN {X 0,Y 594.728,Z 455.556,A -85,B 0,C 180,E1 -1045.238,E2 -1045.238} C_VEL
LIN {X 0,Y 594.603,Z 475.882,A -85,B 0,C 180,E1 -1048.136,E2 -1048.136} C_VEL
LIN {X 0,Y 594.518,Z 496.441,A -85,B 0,C 180,E1 -1051.02,E2 -1051.02} C_VEL
LIN {X 0,Y 594.451,Z 515.958,A -85,B 0,C 180,E1 -1053.691,E2 -1053.691} C_VEL
LIN {X 0,Y 594.767,Z 519.693,A -85,B 0,C 180,E1 -1053.766,E2 -1053.766} C_VEL
LIN {X 0,Y 594.662,Z 624.502,A -85,B 0,C 180,E1 -1055.054,E2 -1055.054} C_VEL
LIN {X 0,Y 594.62,Z 638.594,A -85,B 0,C 180,E1 -1055.384,E2 -1055.384} C_VEL
LIN {X 0,Y 594.585,Z 650.358,A -85,B 0,C 180,E1 -1055.795,E2 -1055.795} C_VEL
LIN {X 0,Y 594.511,Z 661.367,A -85,B 0,C 180,E1 -1056.301,E2 -1056.301} C_VEL
LIN {X 0,Y 594.452,Z 672.344,A -85,B 0,C 180,E1 -1056.945,E2 -1056.945} C_VEL
LIN {X 0,Y 594.416,Z 683.509,A -85,B 0,C 180,E1 -1057.769,E2 -1057.769} C_VEL
LIN {X 0,Y 594.36,Z 693.308,A -85,B 0,C 180,E1 -1058.665,E2 -1058.665} C_VEL
LIN {X 0,Y 594.312,Z 701.427,A -85,B 0,C 180,E1 -1059.583,E2 -1059.583} C_VEL
LIN {X 0,Y 594.301,Z 709.183,A -85,B 0,C 180,E1 -1060.664,E2 -1060.664} C_VEL
LIN {X 0,Y 594.265,Z 715.312,A -85,B 0,C 180,E1 -1061.736,E2 -1061.736} C_VEL
LIN {X 0,Y 594.263,Z 720.036,A -85,B 0,C 180,E1 -1062.803,E2 -1062.803} C_VEL
LIN {X 0,Y 594.249,Z 722.51,A -85,B 0,C 180,E1 -1063.511,E2 -1063.511} C_VEL
LIN {X 0,Y 594.255,Z 724.507,A -85,B 0,C 180,E1 -1064.216,E2 -1064.216} C_VEL
LIN {X 0,Y 594.211,Z 726.039,A -85,B 0,C 180,E1 -1064.918,E2 -1064.918} C_VEL
LIN {X 0,Y 594.259,Z 727.754,A -85,B 0,C 180,E1 -1066.318,E2 -1066.318} C_VEL
LIN {X 0,Y 594.244,Z 727.998,A -85,B 0,C 180,E1 -1067.014,E2 -1067.014} C_VEL
LIN {X 0,Y 594.24,Z 727.796,A -85,B 0,C 180,E1 -1067.709,E2 -1067.709} C_VEL
LIN {X 0,Y 594.252,Z 726.182,A -85,B 0,C 180,E1 -1069.093,E2 -1069.093} C_VEL
LIN {X 0,Y 594.232,Z 724.746,A -85,B 0,C 180,E1 -1069.782,E2 -1069.782} C_VEL
LIN {X 0,Y 594.264,Z 721.763,A -85,B 0,C 180,E1 -1070.813,E2 -1070.813} C_VEL
LIN {X 0,Y 594.28,Z 717.729,A -85,B 0,C 180,E1 -1071.842,E2 -1071.842} C_VEL
LIN {X 0,Y 594.307,Z 711.561,A -85,B 0,C 180,E1 -1073.038,E2 -1073.038} C_VEL
LIN {X 0,Y 594.319,Z 703.592,A -85,B 0,C 180,E1 -1074.231,E2 -1074.231} C_VEL
LIN {X 0,Y 594.343,Z 694.948,A -85,B 0,C 180,E1 -1075.252,E2 -1075.252} C_VEL
LIN {X 0,Y 594.405,Z 686.112,A -85,B 0,C 180,E1 -1076.102,E2 -1076.102} C_VEL
LIN {X 0,Y 594.468,Z 676.428,A -85,B 0,C 180,E1 -1076.866,E2 -1076.866} C_VEL
LIN {X 0,Y 594.504,Z 665.847,A -85,B 0,C 180,E1 -1077.544,E2 -1077.544} C_VEL
LIN {X 0,Y 594.546,Z 654.081,A -85,B 0,C 180,E1 -1078.137,E2 -1078.137} C_VEL
LIN {X 0,Y 594.614,Z 641.854,A -85,B 0,C 180,E1 -1078.603,E2 -1078.603} C_VEL
LIN {X 0,Y 594.679,Z 629.295,A -85,B 0,C 180,E1 -1078.942,E2 -1078.942} C_VEL
LIN {X 0,Y 594.703,Z 614.531,A -85,B 0,C 180,E1 -1079.175,E2 -1079.175} C_VEL
LIN {X 0,Y 594.674,Z 517.746,A -85,B 0,C 180,E1 -1080.349,E2 -1080.349} C_VEL
LIN {X 0,Y 594.418,Z 515.693,A -85,B 0,C 180,E1 -1080.424,E2 -1080.424} C_VEL
LIN {X 0,Y 594.522,Z 496.689,A -85,B 0,C 180,E1 -1083.05,E2 -1083.05} C_VEL
LIN {X 0,Y 594.611,Z 476.188,A -85,B 0,C 180,E1 -1085.936,E2 -1085.936} C_VEL
LIN {X 0,Y 594.717,Z 457.113,A -85,B 0,C 180,E1 -1088.666,E2 -1088.666} C_VEL
LIN {X 0,Y 594.541,Z 451.232,A -85,B 0,C 180,E1 -1089.526,E2 -1089.526} C_VEL
LIN {X 0,Y 594.39,Z 450.481,A -85,B 0,C 180,E1 -1089.7,E2 -1089.7} C_VEL
LIN {X 0,Y 594.35,Z 450.446,A -85,B 0,C 180,E1 -1092.289,E2 -1092.289} C_VEL
LIN {X 0,Y 594.352,Z 450.454,A -85,B 0,C 180,E1 -1095.079,E2 -1095.079} C_VEL
LIN {X 0,Y 594.376,Z 450.451,A -85,B 0,C 180,E1 -1097.194,E2 -1097.194} C_VEL
LIN {X 0,Y 594.359,Z 450.444,A -85,B 0,C 180,E1 -1100.055,E2 -1100.055} C_VEL
LIN {X 0,Y 594.358,Z 450.454,A -85,B 0,C 180,E1 -1102.968,E2 -1102.968} C_VEL
LIN {X 0,Y 594.381,Z 450.447,A -85,B 0,C 180,E1 -1105.193,E2 -1105.193} C_VEL
LIN {X 0,Y 594.376,Z 450.443,A -85,B 0,C 180,E1 -1107.523,E2 -1107.523} C_VEL
LIN {X 0,Y 594.378,Z 450.444,A -85,B 0,C 180,E1 -1110.325,E2 -1110.325} C_VEL
LIN {X 0,Y 594.385,Z 450.447,A -85,B 0,C 180,E1 -1112.95,E2 -1112.95} C_VEL
LIN {X 0,Y 594.36,Z 450.444,A -85,B 0,C 180,E1 -1115.409,E2 -1115.409} C_VEL
LIN {X 0,Y 594.39,Z 450.441,A -85,B 0,C 180,E1 -1117.941,E2 -1117.941} C_VEL
LIN {X 0,Y 594.38,Z 450.446,A -85,B 0,C 180,E1 -1120.821,E2 -1120.821} C_VEL
LIN {X 0,Y 594.373,Z 450.442,A -85,B 0,C 180,E1 -1123.299,E2 -1123.299} C_VEL
LIN {X 0,Y 594.367,Z 450.449,A -85,B 0,C 180,E1 -1126.161,E2 -1126.161} C_VEL
LIN {X 0,Y 594.381,Z 450.448,A -85,B 0,C 180,E1 -1128.535,E2 -1128.535} C_VEL
LIN {X 0,Y 594.377,Z 450.44,A -85,B 0,C 180,E1 -1131.297,E2 -1131.297} C_VEL
LIN {X 0,Y 594.356,Z 450.447,A -85,B 0,C 180,E1 -1133.755,E2 -1133.755} C_VEL
LIN {X 0,Y 594.368,Z 450.452,A -85,B 0,C 180,E1 -1136.237,E2 -1136.237} C_VEL
LIN {X 0,Y 594.366,Z 450.445,A -85,B 0,C 180,E1 -1138.649,E2 -1138.649} C_VEL
LIN {X 0,Y 594.379,Z 450.442,A -85,B 0,C 180,E1 -1141.043,E2 -1141.043} C_VEL
LIN {X 0,Y 594.386,Z 450.65,A -85,B 0,C 180,E1 -1143.444,E2 -1143.444} C_VEL
LIN {X 0,Y 595.216,Z 455.093,A -85,B 0,C 180,E1 -1143.995,E2 -1143.995} C_VEL
LIN {X 0,Y 595.015,Z 479.615,A -85,B 0,C 180,E1 -1146.69,E2 -1146.69} C_VEL
LIN {X 0,Y 594.841,Z 506.619,A -85,B 0,C 180,E1 -1149.601,E2 -1149.601} C_VEL
LIN {X 0,Y 594.66,Z 533.622,A -85,B 0,C 180,E1 -1152.459,E2 -1152.459} C_VEL
LIN {X 0,Y 594.542,Z 560.626,A -85,B 0,C 180,E1 -1155.276,E2 -1155.276} C_VEL
LIN {X 0,Y 594.554,Z 574.079,A -85,B 0,C 180,E1 -1156.64,E2 -1156.64} C_VEL
LIN {X 0,Y 594.755,Z 579.633,A -85,B 0,C 180,E1 -1156.72,E2 -1156.72} C_VEL
LIN {X 0,Y 594.662,Z 683.891,A -85,B 0,C 180,E1 -1157.998,E2 -1157.998} C_VEL
LIN {X 0,Y 594.635,Z 697.18,A -85,B 0,C 180,E1 -1158.3,E2 -1158.3} C_VEL
LIN {X 0,Y 594.597,Z 709.556,A -85,B 0,C 180,E1 -1158.718,E2 -1158.718} C_VEL
LIN {X 0,Y 594.537,Z 721.613,A -85,B 0,C 180,E1 -1159.269,E2 -1159.269} C_VEL
LIN {X 0,Y 594.474,Z 733.184,A -85,B 0,C 180,E1 -1159.956,E2 -1159.956} C_VEL
LIN {X 0,Y 594.414,Z 743.583,A -85,B 0,C 180,E1 -1160.729,E2 -1160.729} C_VEL
LIN {X 0,Y 594.366,Z 752.101,A -85,B 0,C 180,E1 -1161.499,E2 -1161.499} C_VEL
LIN {X 0,Y 594.348,Z 759.951,A -85,B 0,C 180,E1 -1162.354,E2 -1162.354} C_VEL
LIN {X 0,Y 594.284,Z 767.808,A -85,B 0,C 180,E1 -1163.408,E2 -1163.408} C_VEL
LIN {X 0,Y 594.289,Z 774.675,A -85,B 0,C 180,E1 -1164.57,E2 -1164.57} C_VEL
LIN {X 0,Y 594.271,Z 779.367,A -85,B 0,C 180,E1 -1165.59,E2 -1165.59} C_VEL
LIN {X 0,Y 594.267,Z 782.953,A -85,B 0,C 180,E1 -1166.609,E2 -1166.609} C_VEL
LIN {X 0,Y 594.226,Z 784.806,A -85,B 0,C 180,E1 -1167.287,E2 -1167.287} C_VEL
LIN {X 0,Y 594.241,Z 786.2,A -85,B 0,C 180,E1 -1167.966,E2 -1167.966} C_VEL
LIN {X 0,Y 594.239,Z 787.783,A -85,B 0,C 180,E1 -1169.321,E2 -1169.321} C_VEL
LIN {X 0,Y 594.236,Z 788,A -85,B 0,C 180,E1 -1169.999,E2 -1169.999} C_VEL
LIN {X 0,Y 594.247,Z 787.186,A -85,B 0,C 180,E1 -1171.354,E2 -1171.354} C_VEL
LIN {X 0,Y 594.241,Z 786.204,A -85,B 0,C 180,E1 -1172.032,E2 -1172.032} C_VEL
LIN {X 0,Y 594.226,Z 784.812,A -85,B 0,C 180,E1 -1172.71,E2 -1172.71} C_VEL
LIN {X 0,Y 594.289,Z 781.9,A -85,B 0,C 180,E1 -1173.728,E2 -1173.728} C_VEL
LIN {X 0,Y 594.241,Z 777.955,A -85,B 0,C 180,E1 -1174.748,E2 -1174.748} C_VEL
LIN {X 0,Y 594.304,Z 771.884,A -85,B 0,C 180,E1 -1175.938,E2 -1175.938} C_VEL
LIN {X 0,Y 594.311,Z 765.245,A -85,B 0,C 180,E1 -1176.961,E2 -1176.961} C_VEL
LIN {X 0,Y 594.359,Z 757,A -85,B 0,C 180,E1 -1177.985,E2 -1177.985} C_VEL
LIN {X 0,Y 594.382,Z 748.551,A -85,B 0,C 180,E1 -1178.841,E2 -1178.841} C_VEL
LIN {X 0,Y 594.427,Z 738.11,A -85,B 0,C 180,E1 -1179.698,E2 -1179.698} C_VEL
LIN {X 0,Y 594.493,Z 727.779,A -85,B 0,C 180,E1 -1180.385,E2 -1180.385} C_VEL
LIN {X 0,Y 594.561,Z 716.689,A -85,B 0,C 180,E1 -1180.975,E2 -1180.975} C_VEL
LIN {X 0,Y 594.599,Z 704.73,A -85,B 0,C 180,E1 -1181.463,E2 -1181.463} C_VEL
LIN {X 0,Y 594.644,Z 691.404,A -85,B 0,C 180,E1 -1181.849,E2 -1181.849} C_VEL
LIN {X 0,Y 594.692,Z 678.178,A -85,B 0,C 180,E1 -1182.086,E2 -1182.086} C_VEL
LIN {X 0,Y 594.605,Z 574.603,A -85,B 0,C 180,E1 -1183.346,E2 -1183.346} C_VEL
LIN {X 0,Y 594.48,Z 573.359,A -85,B 0,C 180,E1 -1183.414,E2 -1183.414} C_VEL
LIN {X 0,Y 594.601,Z 547.279,A -85,B 0,C 180,E1 -1186.125,E2 -1186.125} C_VEL
LIN {X 0,Y 594.742,Z 519.012,A -85,B 0,C 180,E1 -1189.108,E2 -1189.108} C_VEL
LIN {X 0,Y 594.919,Z 493.487,A -85,B 0,C 180,E1 -1191.845,E2 -1191.845} C_VEL
LIN {X 0,Y 595.156,Z 466.437,A -85,B 0,C 180,E1 -1194.8,E2 -1194.8} C_VEL
LIN {X 0,Y 595.226,Z 453.965,A -85,B 0,C 180,E1 -1196.187,E2 -1196.187} C_VEL
LIN {X 0,Y 594.379,Z 450.564,A -85,B 0,C 180,E1 -1196.639,E2 -1196.639} C_VEL
LIN {X 0,Y 594.366,Z 450.443,A -85,B 0,C 180,E1 -1198.998,E2 -1198.998} C_VEL
LIN {X 0,Y 594.364,Z 450.446,A -85,B 0,C 180,E1 -1201.64,E2 -1201.64} C_VEL
LIN {X 0,Y 594.362,Z 450.453,A -85,B 0,C 180,E1 -1204.135,E2 -1204.135} C_VEL
LIN {X 0,Y 594.323,Z 450.447,A -85,B 0,C 180,E1 -1207.089,E2 -1207.089} C_VEL
LIN {X 0,Y 594.336,Z 450.449,A -85,B 0,C 180,E1 -1209.769,E2 -1209.769} C_VEL
LIN {X 0,Y 594.36,Z 450.45,A -85,B 0,C 180,E1 -1212.374,E2 -1212.374} C_VEL
LIN {X 0,Y 594.327,Z 450.447,A -85,B 0,C 180,E1 -1215.193,E2 -1215.193} C_VEL
LIN {X 0,Y 594.364,Z 450.451,A -85,B 0,C 180,E1 -1218.151,E2 -1218.151} C_VEL
LIN {X 0,Y 594.354,Z 450.443,A -85,B 0,C 180,E1 -1221.192,E2 -1221.192} C_VEL
LIN {X 0,Y 594.333,Z 450.448,A -85,B 0,C 180,E1 -1223.754,E2 -1223.754} C_VEL
LIN {X 0,Y 594.368,Z 450.451,A -85,B 0,C 180,E1 -1226.238,E2 -1226.238} C_VEL
LIN {X 0,Y 594.374,Z 450.446,A -85,B 0,C 180,E1 -1228.65,E2 -1228.65} C_VEL
LIN {X 0,Y 594.362,Z 450.443,A -85,B 0,C 180,E1 -1231.043,E2 -1231.043} C_VEL
LIN {X 0,Y 594.365,Z 450.442,A -85,B 0,C 180,E1 -1233.299,E2 -1233.299} C_VEL
LIN {X 0,Y 594.337,Z 450.446,A -85,B 0,C 180,E1 -1235.573,E2 -1235.573} C_VEL
LIN {X 0,Y 594.348,Z 450.453,A -85,B 0,C 180,E1 -1238.496,E2 -1238.496} C_VEL
LIN {X 0,Y 594.352,Z 450.443,A -85,B 0,C 180,E1 -1241.381,E2 -1241.381} C_VEL
LIN {X 0,Y 594.353,Z 450.45,A -85,B 0,C 180,E1 -1244.218,E2 -1244.218} C_VEL
LIN {X 0,Y 594.347,Z 450.446,A -85,B 0,C 180,E1 -1247.016,E2 -1247.016} C_VEL
LIN {X 0,Y 594.38,Z 450.441,A -85,B 0,C 180,E1 -1249.095,E2 -1249.095} C_VEL
LIN {X 0,Y 594.363,Z 450.443,A -85,B 0,C 180,E1 -1251.842,E2 -1251.842} C_VEL
LIN {X 0,Y 594.388,Z 450.449,A -85,B 0,C 180,E1 -1254.572,E2 -1254.572} C_VEL
LIN {X 0,Y 594.387,Z 450.44,A -85,B 0,C 180,E1 -1257.289,E2 -1257.289} C_VEL
LIN {X 0,Y 594.385,Z 450.441,A -85,B 0,C 180,E1 -1260,E2 -1260} C_VEL
LIN {X 0,Y 594.411,Z 450.444,A -85,B 0,C 180,E1 -1262.71,E2 -1262.71} C_VEL
LIN {X 0,Y 594.377,Z 450.441,A -85,B 0,C 180,E1 -1265.428,E2 -1265.428} C_VEL
LIN {X 0,Y 594.398,Z 450.441,A -85,B 0,C 180,E1 -1268.157,E2 -1268.157} C_VEL
LIN {X 0,Y 594.387,Z 450.442,A -85,B 0,C 180,E1 -1271.08,E2 -1271.08} C_VEL
LIN {X 0,Y 594.368,Z 450.441,A -85,B 0,C 180,E1 -1273.679,E2 -1273.679} C_VEL
LIN {X 0,Y 594.351,Z 450.445,A -85,B 0,C 180,E1 -1275.345,E2 -1275.345} C_VEL
LIN {X 0,Y 593.675,Z 450.529,A -85,B 0,C 180,E1 -1275.91,E2 -1275.91} C_VEL
LIN {X 0,Y 590.806,Z 450.893,A -85,B 0,C 180,E1 -1276.829,E2 -1276.829} C_VEL
LIN {X 0,Y 588.397,Z 451.19,A -85,B 0,C 180,E1 -1277.567,E2 -1277.567} C_VEL
LIN {X 0,Y 587.377,Z 451.315,A -85,B 0,C 180,E1 -1278.137,E2 -1278.137} C_VEL
LIN {X 0,Y 587.302,Z 451.324,A -85,B 0,C 180,E1 -1278.33,E2 -1278.33} C_VEL
LIN {X 0,Y 587.344,Z 451.321,A -85,B 0,C 180,E1 -1281.045,E2 -1281.045} C_VEL
LIN {X 0,Y 587.321,Z 451.32,A -85,B 0,C 180,E1 -1284.007,E2 -1284.007} C_VEL
LIN {X 0,Y 587.326,Z 451.322,A -85,B 0,C 180,E1 -1286.279,E2 -1286.279} C_VEL
LIN {X 0,Y 587.34,Z 451.321,A -85,B 0,C 180,E1 -1289.135,E2 -1289.135} C_VEL
LIN {X 0,Y 587.342,Z 451.317,A -85,B 0,C 180,E1 -1291.838,E2 -1291.838} C_VEL
LIN {X 0,Y 587.346,Z 451.319,A -85,B 0,C 180,E1 -1294.35,E2 -1294.35} C_VEL
LIN {X 0,Y 587.339,Z 451.327,A -85,B 0,C 180,E1 -1296.747,E2 -1296.747} C_VEL
LIN {X 0,Y 587.335,Z 451.32,A -85,B 0,C 180,E1 -1299.36,E2 -1299.36} C_VEL
LIN {X 0,Y 587.322,Z 451.32,A -85,B 0,C 180,E1 -1302.109,E2 -1302.109} C_VEL
LIN {X 0,Y 587.305,Z 451.328,A -85,B 0,C 180,E1 -1305.09,E2 -1305.09} C_VEL
LIN {X 0,Y 587.342,Z 451.317,A -85,B 0,C 180,E1 -1307.929,E2 -1307.929} C_VEL
LIN {X 0,Y 587.337,Z 451.323,A -85,B 0,C 180,E1 -1310.642,E2 -1310.642} C_VEL
LIN {X 0,Y 587.344,Z 451.321,A -85,B 0,C 180,E1 -1313.293,E2 -1313.293} C_VEL
LIN {X 0,Y 587.358,Z 451.315,A -85,B 0,C 180,E1 -1315.781,E2 -1315.781} C_VEL
LIN {X 0,Y 587.348,Z 451.317,A -85,B 0,C 180,E1 -1318.233,E2 -1318.233} C_VEL
LIN {X 0,Y 587.344,Z 451.325,A -85,B 0,C 180,E1 -1320.867,E2 -1320.867} C_VEL
LIN {X 0,Y 587.353,Z 451.316,A -85,B 0,C 180,E1 -1323.82,E2 -1323.82} C_VEL
LIN {X 0,Y 587.331,Z 451.318,A -85,B 0,C 180,E1 -1325.995,E2 -1325.995} C_VEL
LIN {X 0,Y 587.318,Z 451.32,A -85,B 0,C 180,E1 -1328.227,E2 -1328.227} C_VEL
LIN {X 0,Y 587.347,Z 451.326,A -85,B 0,C 180,E1 -1331.153,E2 -1331.153} C_VEL
LIN {X 0,Y 587.324,Z 451.319,A -85,B 0,C 180,E1 -1334.026,E2 -1334.026} C_VEL
LIN {X 0,Y 587.357,Z 451.315,A -85,B 0,C 180,E1 -1336.156,E2 -1336.156} C_VEL
LIN {X 0,Y 587.344,Z 451.324,A -85,B 0,C 180,E1 -1338.964,E2 -1338.964} C_VEL
LIN {X 0,Y 587.368,Z 451.316,A -85,B 0,C 180,E1 -1341.746,E2 -1341.746} C_VEL
LIN {X 0,Y 587.359,Z 451.317,A -85,B 0,C 180,E1 -1344.508,E2 -1344.508} C_VEL
LIN {X 0,Y 587.374,Z 451.323,A -85,B 0,C 180,E1 -1347.258,E2 -1347.258} C_VEL
LIN {X 0,Y 587.384,Z 451.318,A -85,B 0,C 180,E1 -1350.001,E2 -1350.001} C_VEL
LIN {X 0,Y 587.412,Z 451.53,A -85,B 0,C 180,E1 -1350.772,E2 -1350.772} C_VEL
LIN {X 0,Y 587.64,Z 452.671,A -85,B 0,C 180,E1 -1350.879,E2 -1350.879} C_VEL
LIN {X 0,Y 587.848,Z 457.008,A -85,B 0,C 180,E1 -1350.943,E2 -1350.943} C_VEL
LIN {X 0,Y 587.77,Z 534.254,A -85,B 0,C 180,E1 -1351.907,E2 -1351.907} C_VEL
LIN {X 0,Y 587.657,Z 547.296,A -85,B 0,C 180,E1 -1352.207,E2 -1352.207} C_VEL
LIN {X 0,Y 587.609,Z 560.344,A -85,B 0,C 180,E1 -1352.658,E2 -1352.658} C_VEL
LIN {X 0,Y 587.542,Z 571.383,A -85,B 0,C 180,E1 -1353.173,E2 -1353.173} C_VEL
LIN {X 0,Y 587.464,Z 582.881,A -85,B 0,C 180,E1 -1353.86,E2 -1353.86} C_VEL
LIN {X 0,Y 587.38,Z 593.246,A -85,B 0,C 180,E1 -1354.634,E2 -1354.634} C_VEL
LIN {X 0,Y 587.338,Z 602.633,A -85,B 0,C 180,E1 -1355.494,E2 -1355.494} C_VEL
LIN {X 0,Y 587.266,Z 610.851,A -85,B 0,C 180,E1 -1356.419,E2 -1356.419} C_VEL
LIN {X 0,Y 587.239,Z 619.057,A -85,B 0,C 180,E1 -1357.566,E2 -1357.566} C_VEL
LIN {X 0,Y 587.211,Z 624.966,A -85,B 0,C 180,E1 -1358.605,E2 -1358.605} C_VEL
LIN {X 0,Y 587.167,Z 629.64,A -85,B 0,C 180,E1 -1359.648,E2 -1359.648} C_VEL
LIN {X 0,Y 587.183,Z 633.2,A -85,B 0,C 180,E1 -1360.692,E2 -1360.692} C_VEL
LIN {X 0,Y 587.154,Z 635.747,A -85,B 0,C 180,E1 -1361.742,E2 -1361.742} C_VEL
LIN {X 0,Y 587.159,Z 636.919,A -85,B 0,C 180,E1 -1362.443,E2 -1362.443} C_VEL
LIN {X 0,Y 587.145,Z 637.64,A -85,B 0,C 180,E1 -1363.147,E2 -1363.147} C_VEL
LIN {X 0,Y 587.158,Z 637.975,A -85,B 0,C 180,E1 -1364.181,E2 -1364.181} C_VEL
LIN {X 0,Y 587.123,Z 637.352,A -85,B 0,C 180,E1 -1365.27,E2 -1365.27} C_VEL
LIN {X 0,Y 587.137,Z 636.396,A -85,B 0,C 180,E1 -1365.981,E2 -1365.981} C_VEL
LIN {X 0,Y 587.144,Z 634.903,A -85,B 0,C 180,E1 -1366.748,E2 -1366.748} C_VEL
LIN {X 0,Y 587.161,Z 632.042,A -85,B 0,C 180,E1 -1367.773,E2 -1367.773} C_VEL
LIN {X 0,Y 587.179,Z 627.31,A -85,B 0,C 180,E1 -1368.994,E2 -1368.994} C_VEL
LIN {X 0,Y 587.203,Z 621.46,A -85,B 0,C 180,E1 -1370.128,E2 -1370.128} C_VEL
LIN {X 0,Y 587.238,Z 614.273,A -85,B 0,C 180,E1 -1371.226,E2 -1371.226} C_VEL
LIN {X 0,Y 587.292,Z 606.834,A -85,B 0,C 180,E1 -1372.146,E2 -1372.146} C_VEL
LIN {X 0,Y 587.38,Z 596.889,A -85,B 0,C 180,E1 -1373.141,E2 -1373.141} C_VEL
LIN {X 0,Y 587.417,Z 586.174,A -85,B 0,C 180,E1 -1374.004,E2 -1374.004} C_VEL
LIN {X 0,Y 587.509,Z 575.661,A -85,B 0,C 180,E1 -1374.682,E2 -1374.682} C_VEL
LIN {X 0,Y 587.583,Z 563.045,A -85,B 0,C 180,E1 -1375.316,E2 -1375.316} C_VEL
LIN {X 0,Y 587.651,Z 550.509,A -85,B 0,C 180,E1 -1375.788,E2 -1375.788} C_VEL
LIN {X 0,Y 587.736,Z 537.724,A -85,B 0,C 180,E1 -1376.117,E2 -1376.117} C_VEL
LIN {X 0,Y 587.774,Z 519.808,A -85,B 0,C 180,E1 -1376.378,E2 -1376.378} C_VEL
LIN {X 0,Y 587.76,Z 453.008,A -85,B 0,C 180,E1 -1377.2,E2 -1377.2} C_VEL
LIN {X 0,Y 587.422,Z 451.648,A -85,B 0,C 180,E1 -1377.294,E2 -1377.294} C_VEL
LIN {X 0,Y 587.358,Z 451.333,A -85,B 0,C 180,E1 -1377.429,E2 -1377.429} C_VEL
LIN {X 0,Y 587.334,Z 451.321,A -85,B 0,C 180,E1 -1380.171,E2 -1380.171} C_VEL
LIN {X 0,Y 587.341,Z 451.324,A -85,B 0,C 180,E1 -1383.112,E2 -1383.112} C_VEL
LIN {X 0,Y 587.293,Z 451.324,A -85,B 0,C 180,E1 -1385.901,E2 -1385.901} C_VEL
LIN {X 0,Y 587.325,Z 451.324,A -85,B 0,C 180,E1 -1388.481,E2 -1388.481} C_VEL
LIN {X 0,Y 587.338,Z 451.323,A -85,B 0,C 180,E1 -1391.158,E2 -1391.158} C_VEL
LIN {X 0,Y 587.316,Z 451.321,A -85,B 0,C 180,E1 -1394.113,E2 -1394.113} C_VEL
LIN {X 0,Y 587.316,Z 451.329,A -85,B 0,C 180,E1 -1396.994,E2 -1396.994} C_VEL
LIN {X 0,Y 587.311,Z 451.322,A -85,B 0,C 180,E1 -1399.746,E2 -1399.746} C_VEL
LIN {X 0,Y 587.345,Z 451.321,A -85,B 0,C 180,E1 -1402.393,E2 -1402.393} C_VEL
LIN {X 0,Y 587.381,Z 451.528,A -85,B 0,C 180,E1 -1404.34,E2 -1404.34} C_VEL
LIN {X 0,Y 587.828,Z 455.629,A -85,B 0,C 180,E1 -1404.979,E2 -1404.979} C_VEL
LIN {X 0,Y 587.677,Z 474.118,A -85,B 0,C 180,E1 -1407.651,E2 -1407.651} C_VEL
LIN {X 0,Y 587.53,Z 495.071,A -85,B 0,C 180,E1 -1410.631,E2 -1410.631} C_VEL
LIN {X 0,Y 587.421,Z 515.339,A -85,B 0,C 180,E1 -1413.467,E2 -1413.467} C_VEL
LIN {X 0,Y 587.521,Z 516.837,A -85,B 0,C 180,E1 -1413.561,E2 -1413.561} C_VEL
LIN {X 0,Y 587.883,Z 522.345,A -85,B 0,C 180,E1 -1413.641,E2 -1413.641} C_VEL
LIN {X 0,Y 587.738,Z 624.137,A -85,B 0,C 180,E1 -1414.905,E2 -1414.905} C_VEL
LIN {X 0,Y 587.664,Z 637.367,A -85,B 0,C 180,E1 -1415.209,E2 -1415.209} C_VEL
LIN {X 0,Y 587.611,Z 650.24,A -85,B 0,C 180,E1 -1415.656,E2 -1415.656} C_VEL
LIN {X 0,Y 587.531,Z 661.702,A -85,B 0,C 180,E1 -1416.19,E2 -1416.19} C_VEL
LIN {X 0,Y 587.436,Z 673.028,A -85,B 0,C 180,E1 -1416.869,E2 -1416.869} C_VEL
LIN {X 0,Y 587.398,Z 683.709,A -85,B 0,C 180,E1 -1417.674,E2 -1417.674} C_VEL
LIN {X 0,Y 587.305,Z 693.591,A -85,B 0,C 180,E1 -1418.594,E2 -1418.594} C_VEL
LIN {X 0,Y 587.239,Z 701.555,A -85,B 0,C 180,E1 -1419.509,E2 -1419.509} C_VEL
LIN {X 0,Y 587.219,Z 709.171,A -85,B 0,C 180,E1 -1420.585,E2 -1420.585} C_VEL
LIN {X 0,Y 587.21,Z 714.461,A -85,B 0,C 180,E1 -1421.509,E2 -1421.509} C_VEL
LIN {X 0,Y 587.166,Z 719.403,A -85,B 0,C 180,E1 -1422.589,E2 -1422.589} C_VEL
LIN {X 0,Y 587.154,Z 723.112,A -85,B 0,C 180,E1 -1423.663,E2 -1423.663} C_VEL
LIN {X 0,Y 587.133,Z 725.717,A -85,B 0,C 180,E1 -1424.732,E2 -1424.732} C_VEL
LIN {X 0,Y 587.163,Z 727.342,A -85,B 0,C 180,E1 -1425.821,E2 -1425.821} C_VEL
LIN {X 0,Y 587.146,Z 727.963,A -85,B 0,C 180,E1 -1426.855,E2 -1426.855} C_VEL
LIN {X 0,Y 587.161,Z 727.869,A -85,B 0,C 180,E1 -1427.558,E2 -1427.558} C_VEL
LIN {X 0,Y 587.156,Z 727.352,A -85,B 0,C 180,E1 -1428.26,E2 -1428.26} C_VEL
LIN {X 0,Y 587.17,Z 726.436,A -85,B 0,C 180,E1 -1428.959,E2 -1428.959} C_VEL
LIN {X 0,Y 587.143,Z 725.097,A -85,B 0,C 180,E1 -1429.657,E2 -1429.657} C_VEL
LIN {X 0,Y 587.189,Z 722.267,A -85,B 0,C 180,E1 -1430.702,E2 -1430.702} C_VEL
LIN {X 0,Y 587.19,Z 718.406,A -85,B 0,C 180,E1 -1431.743,E2 -1431.743} C_VEL
LIN {X 0,Y 587.216,Z 713.408,A -85,B 0,C 180,E1 -1432.781,E2 -1432.781} C_VEL
LIN {X 0,Y 587.221,Z 707.143,A -85,B 0,C 180,E1 -1433.817,E2 -1433.817} C_VEL
LIN {X 0,Y 587.305,Z 699.372,A -85,B 0,C 180,E1 -1434.851,E2 -1434.851} C_VEL
LIN {X 0,Y 587.319,Z 691.448,A -85,B 0,C 180,E1 -1435.711,E2 -1435.711} C_VEL
LIN {X 0,Y 587.387,Z 681.834,A -85,B 0,C 180,E1 -1436.571,E2 -1436.571} C_VEL
LIN {X 0,Y 587.476,Z 671.201,A -85,B 0,C 180,E1 -1437.343,E2 -1437.343} C_VEL
LIN {X 0,Y 587.541,Z 660.837,A -85,B 0,C 180,E1 -1437.944,E2 -1437.944} C_VEL
LIN {X 0,Y 587.6,Z 649.679,A -85,B 0,C 180,E1 -1438.458,E2 -1438.458} C_VEL
LIN {X 0,Y 587.703,Z 636.407,A -85,B 0,C 180,E1 -1438.908,E2 -1438.908} C_VEL
LIN {X 0,Y 587.732,Z 624.041,A -85,B 0,C 180,E1 -1439.187,E2 -1439.187} C_VEL
LIN {X 0,Y 587.714,Z 518.054,A -85,B 0,C 180,E1 -1440.506,E2 -1440.506} C_VEL
LIN {X 0,Y 587.384,Z 515.8,A -85,B 0,C 180,E1 -1440.579,E2 -1440.579} C_VEL
LIN {X 0,Y 587.524,Z 497.815,A -85,B 0,C 180,E1 -1443.086,E2 -1443.086} C_VEL
LIN {X 0,Y 587.649,Z 477.313,A -85,B 0,C 180,E1 -1446.007,E2 -1446.007} C_VEL
LIN {X 0,Y 587.791,Z 458.239,A -85,B 0,C 180,E1 -1448.769,E2 -1448.769} C_VEL
LIN {X 0,Y 587.546,Z 452.372,A -85,B 0,C 180,E1 -1449.641,E2 -1449.641} C_VEL
LIN {X 0,Y 587.359,Z 451.354,A -85,B 0,C 180,E1 -1449.861,E2 -1449.861} C_VEL
LIN {X 0,Y 587.305,Z 451.324,A -85,B 0,C 180,E1 -1452.439,E2 -1452.439} C_VEL
LIN {X 0,Y 587.315,Z 451.323,A -85,B 0,C 180,E1 -1454.554,E2 -1454.554} C_VEL
LIN {X 0,Y 587.309,Z 451.327,A -85,B 0,C 180,E1 -1457.407,E2 -1457.407} C_VEL
LIN {X 0,Y 587.308,Z 451.325,A -85,B 0,C 180,E1 -1459.577,E2 -1459.577} C_VEL
LIN {X 0,Y 587.315,Z 451.322,A -85,B 0,C 180,E1 -1461.775,E2 -1461.775} C_VEL
LIN {X 0,Y 587.321,Z 451.328,A -85,B 0,C 180,E1 -1464.76,E2 -1464.76} C_VEL
LIN {X 0,Y 587.349,Z 451.317,A -85,B 0,C 180,E1 -1467.691,E2 -1467.691} C_VEL
LIN {X 0,Y 587.333,Z 451.324,A -85,B 0,C 180,E1 -1470.508,E2 -1470.508} C_VEL
LIN {X 0,Y 587.347,Z 451.321,A -85,B 0,C 180,E1 -1473.111,E2 -1473.111} C_VEL
LIN {X 0,Y 587.306,Z 451.322,A -85,B 0,C 180,E1 -1475.538,E2 -1475.538} C_VEL
LIN {X 0,Y 587.345,Z 451.318,A -85,B 0,C 180,E1 -1477.838,E2 -1477.838} C_VEL
LIN {X 0,Y 587.319,Z 451.326,A -85,B 0,C 180,E1 -1480.254,E2 -1480.254} C_VEL
LIN {X 0,Y 587.321,Z 451.322,A -85,B 0,C 180,E1 -1483.118,E2 -1483.118} C_VEL
LIN {X 0,Y 587.319,Z 451.325,A -85,B 0,C 180,E1 -1486.048,E2 -1486.048} C_VEL
LIN {X 0,Y 587.339,Z 451.32,A -85,B 0,C 180,E1 -1488.925,E2 -1488.925} C_VEL
LIN {X 0,Y 587.327,Z 451.318,A -85,B 0,C 180,E1 -1491.519,E2 -1491.519} C_VEL
LIN {X 0,Y 587.289,Z 451.333,A -85,B 0,C 180,E1 -1494.099,E2 -1494.099} C_VEL
LIN {X 0,Y 587.341,Z 451.319,A -85,B 0,C 180,E1 -1496.888,E2 -1496.888} C_VEL
LIN {X 0,Y 587.335,Z 451.325,A -85,B 0,C 180,E1 -1499.829,E2 -1499.829} C_VEL
LIN {X 0,Y 587.306,Z 451.33,A -85,B 0,C 180,E1 -1502.316,E2 -1502.316} C_VEL
LIN {X 0,Y 587.354,Z 451.565,A -85,B 0,C 180,E1 -1503.207,E2 -1503.207} C_VEL
LIN {X 0,Y 588.387,Z 455.986,A -85,B 0,C 180,E1 -1503.771,E2 -1503.771} C_VEL
LIN {X 0,Y 588.224,Z 476.239,A -85,B 0,C 180,E1 -1506.031,E2 -1506.031} C_VEL
LIN {X 0,Y 588.042,Z 499.572,A -85,B 0,C 180,E1 -1508.589,E2 -1508.589} C_VEL
LIN {X 0,Y 587.816,Z 526.872,A -85,B 0,C 180,E1 -1511.527,E2 -1511.527} C_VEL
LIN {X 0,Y 587.576,Z 552.188,A -85,B 0,C 180,E1 -1514.209,E2 -1514.209} C_VEL
LIN {X 0,Y 587.493,Z 573.851,A -85,B 0,C 180,E1 -1516.465,E2 -1516.465} C_VEL
LIN {X 0,Y 587.899,Z 577.845,A -85,B 0,C 180,E1 -1516.541,E2 -1516.541} C_VEL
LIN {X 0,Y 587.722,Z 683.891,A -85,B 0,C 180,E1 -1517.854,E2 -1517.854} C_VEL
LIN {X 0,Y 587.68,Z 697.181,A -85,B 0,C 180,E1 -1518.16,E2 -1518.16} C_VEL
LIN {X 0,Y 587.629,Z 709.741,A -85,B 0,C 180,E1 -1518.59,E2 -1518.59} C_VEL
LIN {X 0,Y 587.555,Z 721.612,A -85,B 0,C 180,E1 -1519.14,E2 -1519.14} C_VEL
LIN {X 0,Y 587.471,Z 733.185,A -85,B 0,C 180,E1 -1519.836,E2 -1519.836} C_VEL
LIN {X 0,Y 587.393,Z 743.584,A -85,B 0,C 180,E1 -1520.617,E2 -1520.617} C_VEL
LIN {X 0,Y 587.31,Z 752.101,A -85,B 0,C 180,E1 -1521.396,E2 -1521.396} C_VEL
LIN {X 0,Y 587.274,Z 759.951,A -85,B 0,C 180,E1 -1522.262,E2 -1522.262} C_VEL
LIN {X 0,Y 587.231,Z 766.462,A -85,B 0,C 180,E1 -1523.125,E2 -1523.125} C_VEL
LIN {X 0,Y 587.236,Z 772.86,A -85,B 0,C 180,E1 -1524.16,E2 -1524.16} C_VEL
LIN {X 0,Y 587.147,Z 777.945,A -85,B 0,C 180,E1 -1525.193,E2 -1525.193} C_VEL
LIN {X 0,Y 587.213,Z 781.892,A -85,B 0,C 180,E1 -1526.225,E2 -1526.225} C_VEL
LIN {X 0,Y 587.132,Z 784.806,A -85,B 0,C 180,E1 -1527.254,E2 -1527.254} C_VEL
LIN {X 0,Y 587.14,Z 786.199,A -85,B 0,C 180,E1 -1527.941,E2 -1527.941} C_VEL
LIN {X 0,Y 587.14,Z 787.783,A -85,B 0,C 180,E1 -1529.313,E2 -1529.313} C_VEL
LIN {X 0,Y 587.137,Z 788,A -85,B 0,C 180,E1 -1529.999,E2 -1529.999} C_VEL
LIN {X 0,Y 587.147,Z 787.186,A -85,B 0,C 180,E1 -1531.371,E2 -1531.371} C_VEL
LIN {X 0,Y 587.14,Z 786.203,A -85,B 0,C 180,E1 -1532.057,E2 -1532.057} C_VEL
LIN {X 0,Y 587.132,Z 784.812,A -85,B 0,C 180,E1 -1532.743,E2 -1532.743} C_VEL
LIN {X 0,Y 587.213,Z 781.9,A -85,B 0,C 180,E1 -1533.773,E2 -1533.773} C_VEL
LIN {X 0,Y 587.147,Z 777.954,A -85,B 0,C 180,E1 -1534.805,E2 -1534.805} C_VEL
LIN {X 0,Y 587.217,Z 771.885,A -85,B 0,C 180,E1 -1536.01,E2 -1536.01} C_VEL
LIN {X 0,Y 587.246,Z 765.245,A -85,B 0,C 180,E1 -1537.045,E2 -1537.045} C_VEL
LIN {X 0,Y 587.299,Z 757,A -85,B 0,C 180,E1 -1538.082,E2 -1538.082} C_VEL
LIN {X 0,Y 587.343,Z 748.551,A -85,B 0,C 180,E1 -1538.948,E2 -1538.948} C_VEL
LIN {X 0,Y 587.414,Z 738.111,A -85,B 0,C 180,E1 -1539.815,E2 -1539.815} C_VEL
LIN {X 0,Y 587.511,Z 727.779,A -85,B 0,C 180,E1 -1540.51,E2 -1540.51} C_VEL
LIN {X 0,Y 587.582,Z 715.821,A -85,B 0,C 180,E1 -1541.148,E2 -1541.148} C_VEL
LIN {X 0,Y 587.63,Z 703.624,A -85,B 0,C 180,E1 -1541.638,E2 -1541.638} C_VEL
LIN {X 0,Y 587.7,Z 690.49,A -85,B 0,C 180,E1 -1542.013,E2 -1542.013} C_VEL
LIN {X 0,Y 587.772,Z 678.178,A -85,B 0,C 180,E1 -1542.23,E2 -1542.23} C_VEL
LIN {X 0,Y 587.74,Z 575.578,A -85,B 0,C 180,E1 -1543.491,E2 -1543.491} C_VEL
LIN {X 0,Y 587.488,Z 573.589,A -85,B 0,C 180,E1 -1543.555,E2 -1543.555} C_VEL
LIN {X 0,Y 587.668,Z 547.279,A -85,B 0,C 180,E1 -1546.321,E2 -1546.321} C_VEL
LIN {X 0,Y 587.849,Z 519.392,A -85,B 0,C 180,E1 -1549.3,E2 -1549.3} C_VEL
LIN {X 0,Y 588.083,Z 493.487,A -85,B 0,C 180,E1 -1552.112,E2 -1552.112} C_VEL
LIN {X 0,Y 588.375,Z 468.442,A -85,B 0,C 180,E1 -1554.881,E2 -1554.881} C_VEL
LIN {X 0,Y 588.309,Z 455.295,A -85,B 0,C 180,E1 -1556.368,E2 -1556.368} C_VEL
LIN {X 0,Y 587.314,Z 451.404,A -85,B 0,C 180,E1 -1556.901,E2 -1556.901} C_VEL
LIN {X 0,Y 587.306,Z 451.324,A -85,B 0,C 180,E1 -1559.38,E2 -1559.38} C_VEL
LIN {X 0,Y 587.333,Z 451.325,A -85,B 0,C 180,E1 -1561.833,E2 -1561.833} C_VEL
LIN {X 0,Y 587.327,Z 451.326,A -85,B 0,C 180,E1 -1564.344,E2 -1564.344} C_VEL
LIN {X 0,Y 587.308,Z 451.323,A -85,B 0,C 180,E1 -1567.609,E2 -1567.609} C_VEL
LIN {X 0,Y 587.299,Z 451.332,A -85,B 0,C 180,E1 -1570.254,E2 -1570.254} C_VEL
LIN {X 0,Y 587.293,Z 451.323,A -85,B 0,C 180,E1 -1573.116,E2 -1573.116} C_VEL
LIN {X 0,Y 587.303,Z 451.329,A -85,B 0,C 180,E1 -1576.047,E2 -1576.047} C_VEL
LIN {X 0,Y 587.322,Z 451.32,A -85,B 0,C 180,E1 -1578.924,E2 -1578.924} C_VEL
LIN {X 0,Y 587.304,Z 451.322,A -85,B 0,C 180,E1 -1581.518,E2 -1581.518} C_VEL
LIN {X 0,Y 587.276,Z 451.332,A -85,B 0,C 180,E1 -1584.099,E2 -1584.099} C_VEL
LIN {X 0,Y 587.322,Z 451.325,A -85,B 0,C 180,E1 -1586.602,E2 -1586.602} C_VEL
LIN {X 0,Y 587.32,Z 451.32,A -85,B 0,C 180,E1 -1589.033,E2 -1589.033} C_VEL
LIN {X 0,Y 587.297,Z 451.322,A -85,B 0,C 180,E1 -1591.401,E2 -1591.401} C_VEL
LIN {X 0,Y 587.319,Z 451.322,A -85,B 0,C 180,E1 -1593.824,E2 -1593.824} C_VEL
LIN {X 0,Y 587.294,Z 451.327,A -85,B 0,C 180,E1 -1595.991,E2 -1595.991} C_VEL
LIN {X 0,Y 587.317,Z 451.322,A -85,B 0,C 180,E1 -1598.962,E2 -1598.962} C_VEL
LIN {X 0,Y 587.326,Z 451.319,A -85,B 0,C 180,E1 -1601.15,E2 -1601.15} C_VEL
LIN {X 0,Y 587.303,Z 451.325,A -85,B 0,C 180,E1 -1604.024,E2 -1604.024} C_VEL
LIN {X 0,Y 587.298,Z 451.326,A -85,B 0,C 180,E1 -1606.858,E2 -1606.858} C_VEL
LIN {X 0,Y 587.38,Z 451.315,A -85,B 0,C 180,E1 -1608.963,E2 -1608.963} C_VEL
LIN {X 0,Y 587.367,Z 451.324,A -85,B 0,C 180,E1 -1612.437,E2 -1612.437} C_VEL
LIN {X 0,Y 587.342,Z 451.318,A -85,B 0,C 180,E1 -1615.195,E2 -1615.195} C_VEL
LIN {X 0,Y 587.34,Z 451.319,A -85,B 0,C 180,E1 -1617.943,E2 -1617.943} C_VEL
LIN {X 0,Y 587.391,Z 451.319,A -85,B 0,C 180,E1 -1620.685,E2 -1620.685} C_VEL
LIN {X 0,Y 587.316,Z 451.32,A -85,B 0,C 180,E1 -1623.43,E2 -1623.43} C_VEL
LIN {X 0,Y 587.341,Z 451.317,A -85,B 0,C 180,E1 -1625.493,E2 -1625.493} C_VEL
LIN {X 0,Y 587.354,Z 451.32,A -85,B 0,C 180,E1 -1628.255,E2 -1628.255} C_VEL
LIN {X 0,Y 587.348,Z 451.319,A -85,B 0,C 180,E1 -1631.141,E2 -1631.141} C_VEL
LIN {X 0,Y 587.35,Z 451.32,A -85,B 0,C 180,E1 -1634.261,E2 -1634.261} C_VEL
LIN {X 0,Y 587.339,Z 451.318,A -85,B 0,C 180,E1 -1637.406,E2 -1637.406} C_VEL
LIN {X 0,Y 587.302,Z 451.324,A -85,B 0,C 180,E1 -1638.33,E2 -1638.33} C_VEL
LIN {X 0,Y 586.662,Z 451.41,A -85,B 0,C 180,E1 -1638.902,E2 -1638.902} C_VEL
LIN {X 0,Y 583.836,Z 451.761,A -85,B 0,C 180,E1 -1639.831,E2 -1639.831} C_VEL
LIN {X 0,Y 581.423,Z 452.063,A -85,B 0,C 180,E1 -1640.578,E2 -1640.578} C_VEL
LIN {X 0,Y 580.368,Z 452.189,A -85,B 0,C 180,E1 -1641.155,E2 -1641.155} C_VEL
LIN {X 0,Y 580.272,Z 452.199,A -85,B 0,C 180,E1 -1641.35,E2 -1641.35} C_VEL
LIN {X 0,Y 580.286,Z 452.2,A -85,B 0,C 180,E1 -1644.317,E2 -1644.317} C_VEL
LIN {X 0,Y 580.269,Z 452.206,A -85,B 0,C 180,E1 -1646.623,E2 -1646.623} C_VEL
LIN {X 0,Y 580.291,Z 452.197,A -85,B 0,C 180,E1 -1649.311,E2 -1649.311} C_VEL
LIN {X 0,Y 580.29,Z 452.197,A -85,B 0,C 180,E1 -1652.201,E2 -1652.201} C_VEL
LIN {X 0,Y 580.291,Z 452.204,A -85,B 0,C 180,E1 -1654.696,E2 -1654.696} C_VEL
LIN {X 0,Y 580.288,Z 452.199,A -85,B 0,C 180,E1 -1657.269,E2 -1657.269} C_VEL
LIN {X 0,Y 580.287,Z 452.198,A -85,B 0,C 180,E1 -1660.272,E2 -1660.272} C_VEL
LIN {X 0,Y 580.27,Z 452.206,A -85,B 0,C 180,E1 -1662.707,E2 -1662.707} C_VEL
LIN {X 0,Y 580.263,Z 452.199,A -85,B 0,C 180,E1 -1665.609,E2 -1665.609} C_VEL
LIN {X 0,Y 580.31,Z 452.194,A -85,B 0,C 180,E1 -1668.236,E2 -1668.236} C_VEL
LIN {X 0,Y 580.282,Z 452.206,A -85,B 0,C 180,E1 -1670.967,E2 -1670.967} C_VEL
LIN {X 0,Y 580.271,Z 452.199,A -85,B 0,C 180,E1 -1673.598,E2 -1673.598} C_VEL
LIN {X 0,Y 580.31,Z 452.193,A -85,B 0,C 180,E1 -1676.147,E2 -1676.147} C_VEL
LIN {X 0,Y 580.283,Z 452.201,A -85,B 0,C 180,E1 -1678.617,E2 -1678.617} C_VEL
LIN {X 0,Y 580.289,Z 452.206,A -85,B 0,C 180,E1 -1681.025,E2 -1681.025} C_VEL
LIN {X 0,Y 580.286,Z 452.197,A -85,B 0,C 180,E1 -1683.667,E2 -1683.667} C_VEL
LIN {X 0,Y 580.295,Z 452.196,A -85,B 0,C 180,E1 -1685.685,E2 -1685.685} C_VEL
LIN {X 0,Y 580.268,Z 452.198,A -85,B 0,C 180,E1 -1687.949,E2 -1687.949} C_VEL
LIN {X 0,Y 580.314,Z 452.2,A -85,B 0,C 180,E1 -1690.915,E2 -1690.915} C_VEL
LIN {X 0,Y 580.278,Z 452.197,A -85,B 0,C 180,E1 -1693.827,E2 -1693.827} C_VEL
LIN {X 0,Y 580.323,Z 452.191,A -85,B 0,C 180,E1 -1695.984,E2 -1695.984} C_VEL
LIN {X 0,Y 580.301,Z 452.199,A -85,B 0,C 180,E1 -1698.828,E2 -1698.828} C_VEL
LIN {X 0,Y 580.332,Z 452.194,A -85,B 0,C 180,E1 -1701.645,E2 -1701.645} C_VEL
LIN {X 0,Y 580.327,Z 452.192,A -85,B 0,C 180,E1 -1704.441,E2 -1704.441} C_VEL
LIN {X 0,Y 580.34,Z 452.199,A -85,B 0,C 180,E1 -1707.225,E2 -1707.225} C_VEL
LIN {X 0,Y 580.353,Z 452.196,A -85,B 0,C 180,E1 -1710.001,E2 -1710.001} C_VEL
LIN {X 0,Y 580.378,Z 452.444,A -85,B 0,C 180,E1 -1710.63,E2 -1710.63} C_VEL
LIN {X 0,Y 580.6,Z 453.503,A -85,B 0,C 180,E1 -1710.727,E2 -1710.727} C_VEL
LIN {X 0,Y 580.949,Z 456.712,A -85,B 0,C 180,E1 -1710.781,E2 -1710.781} C_VEL
LIN {X 0,Y 580.833,Z 534.08,A -85,B 0,C 180,E1 -1711.756,E2 -1711.756} C_VEL
LIN {X 0,Y 580.71,Z 547.181,A -85,B 0,C 180,E1 -1712.06,E2 -1712.06} C_VEL
LIN {X 0,Y 580.651,Z 560.262,A -85,B 0,C 180,E1 -1712.516,E2 -1712.516} C_VEL
LIN {X 0,Y 580.557,Z 571.326,A -85,B 0,C 180,E1 -1713.037,E2 -1713.037} C_VEL
LIN {X 0,Y 580.446,Z 582.84,A -85,B 0,C 180,E1 -1713.733,E2 -1713.733} C_VEL
LIN {X 0,Y 580.344,Z 593.217,A -85,B 0,C 180,E1 -1714.516,E2 -1714.516} C_VEL
LIN {X 0,Y 580.295,Z 602.606,A -85,B 0,C 180,E1 -1715.387,E2 -1715.387} C_VEL
LIN {X 0,Y 580.202,Z 611.632,A -85,B 0,C 180,E1 -1716.427,E2 -1716.427} C_VEL
LIN {X 0,Y 580.165,Z 619.039,A -85,B 0,C 180,E1 -1717.484,E2 -1717.484} C_VEL
LIN {X 0,Y 580.11,Z 625.808,A -85,B 0,C 180,E1 -1718.711,E2 -1718.711} C_VEL
LIN {X 0,Y 580.082,Z 630.286,A -85,B 0,C 180,E1 -1719.767,E2 -1719.767} C_VEL
LIN {X 0,Y 580.075,Z 634.334,A -85,B 0,C 180,E1 -1721.078,E2 -1721.078} C_VEL
LIN {X 0,Y 580.053,Z 636.08,A -85,B 0,C 180,E1 -1721.888,E2 -1721.888} C_VEL
LIN {X 0,Y 580.049,Z 637.119,A -85,B 0,C 180,E1 -1722.598,E2 -1722.598} C_VEL
LIN {X 0,Y 580.06,Z 637.758,A -85,B 0,C 180,E1 -1723.31,E2 -1723.31} C_VEL
LIN {X 0,Y 580.049,Z 637.963,A -85,B 0,C 180,E1 -1724.236,E2 -1724.236} C_VEL
LIN {X 0,Y 580.019,Z 637.152,A -85,B 0,C 180,E1 -1725.461,E2 -1725.461} C_VEL
LIN {X 0,Y 580.037,Z 636.109,A -85,B 0,C 180,E1 -1726.182,E2 -1726.182} C_VEL
LIN {X 0,Y 580.041,Z 634.6,A -85,B 0,C 180,E1 -1726.906,E2 -1726.906} C_VEL
LIN {X 0,Y 580.08,Z 631.449,A -85,B 0,C 180,E1 -1727.997,E2 -1727.997} C_VEL
LIN {X 0,Y 580.098,Z 627.124,A -85,B 0,C 180,E1 -1729.095,E2 -1729.095} C_VEL
LIN {X 0,Y 580.118,Z 621.477,A -85,B 0,C 180,E1 -1730.199,E2 -1730.199} C_VEL
LIN {X 0,Y 580.186,Z 614.297,A -85,B 0,C 180,E1 -1731.31,E2 -1731.31} C_VEL
LIN {X 0,Y 580.254,Z 606.863,A -85,B 0,C 180,E1 -1732.242,E2 -1732.242} C_VEL
LIN {X 0,Y 580.357,Z 597.337,A -85,B 0,C 180,E1 -1733.212,E2 -1733.212} C_VEL
LIN {X 0,Y 580.395,Z 587.476,A -85,B 0,C 180,E1 -1734.028,E2 -1734.028} C_VEL
LIN {X 0,Y 580.519,Z 576.313,A -85,B 0,C 180,E1 -1734.773,E2 -1734.773} C_VEL
LIN {X 0,Y 580.615,Z 564.201,A -85,B 0,C 180,E1 -1735.402,E2 -1735.402} C_VEL
LIN {X 0,Y 580.685,Z 550.961,A -85,B 0,C 180,E1 -1735.915,E2 -1735.915} C_VEL
LIN {X 0,Y 580.797,Z 538.567,A -85,B 0,C 180,E1 -1736.247,E2 -1736.247} C_VEL
LIN {X 0,Y 580.829,Z 522.715,A -85,B 0,C 180,E1 -1736.492,E2 -1736.492} C_VEL
LIN {X 0,Y 580.853,Z 454.403,A -85,B 0,C 180,E1 -1737.34,E2 -1737.34} C_VEL
LIN {X 0,Y 580.415,Z 452.774,A -85,B 0,C 180,E1 -1737.415,E2 -1737.415} C_VEL
LIN {X 0,Y 580.313,Z 452.228,A -85,B 0,C 180,E1 -1737.548,E2 -1737.548} C_VEL
LIN {X 0,Y 580.299,Z 452.202,A -85,B 0,C 180,E1 -1740.576,E2 -1740.576} C_VEL
LIN {X 0,Y 580.287,Z 452.2,A -85,B 0,C 180,E1 -1743.314,E2 -1743.314} C_VEL
LIN {X 0,Y 580.248,Z 452.202,A -85,B 0,C 180,E1 -1745.757,E2 -1745.757} C_VEL
LIN {X 0,Y 580.288,Z 452.197,A -85,B 0,C 180,E1 -1748.147,E2 -1748.147} C_VEL
LIN {X 0,Y 580.301,Z 452.205,A -85,B 0,C 180,E1 -1750.844,E2 -1750.844} C_VEL
LIN {X 0,Y 580.277,Z 452.198,A -85,B 0,C 180,E1 -1753.659,E2 -1753.659} C_VEL
LIN {X 0,Y 580.278,Z 452.204,A -85,B 0,C 180,E1 -1756.61,E2 -1756.61} C_VEL
LIN {X 0,Y 580.3,Z 452.2,A -85,B 0,C 180,E1 -1759.157,E2 -1759.157} C_VEL
LIN {X 0,Y 580.289,Z 452.197,A -85,B 0,C 180,E1 -1761.928,E2 -1761.928} C_VEL
LIN {X 0,Y 580.323,Z 452.377,A -85,B 0,C 180,E1 -1764.171,E2 -1764.171} C_VEL
LIN {X 0,Y 580.908,Z 457.127,A -85,B 0,C 180,E1 -1764.924,E2 -1764.924} C_VEL
LIN {X 0,Y 580.7,Z 477.551,A -85,B 0,C 180,E1 -1767.908,E2 -1767.908} C_VEL
LIN {X 0,Y 580.543,Z 496.623,A -85,B 0,C 180,E1 -1770.65,E2 -1770.65} C_VEL
LIN {X 0,Y 580.412,Z 515.662,A -85,B 0,C 180,E1 -1773.335,E2 -1773.335} C_VEL
LIN {X 0,Y 580.642,Z 517.672,A -85,B 0,C 180,E1 -1773.412,E2 -1773.412} C_VEL
LIN {X 0,Y 581.002,Z 522.492,A -85,B 0,C 180,E1 -1773.481,E2 -1773.481} C_VEL
LIN {X 0,Y 580.817,Z 623.763,A -85,B 0,C 180,E1 -1774.753,E2 -1774.753} C_VEL
LIN {X 0,Y 580.772,Z 636.848,A -85,B 0,C 180,E1 -1775.051,E2 -1775.051} C_VEL
LIN {X 0,Y 580.615,Z 649.505,A -85,B 0,C 180,E1 -1775.486,E2 -1775.486} C_VEL
LIN {X 0,Y 580.558,Z 660.181,A -85,B 0,C 180,E1 -1775.981,E2 -1775.981} C_VEL
LIN {X 0,Y 580.449,Z 671.999,A -85,B 0,C 180,E1 -1776.674,E2 -1776.674} C_VEL
LIN {X 0,Y 580.363,Z 682.783,A -85,B 0,C 180,E1 -1777.483,E2 -1777.483} C_VEL
LIN {X 0,Y 580.283,Z 691.943,A -85,B 0,C 180,E1 -1778.322,E2 -1778.322} C_VEL
LIN {X 0,Y 580.218,Z 700.435,A -85,B 0,C 180,E1 -1779.273,E2 -1779.273} C_VEL
LIN {X 0,Y 580.177,Z 708.333,A -85,B 0,C 180,E1 -1780.376,E2 -1780.376} C_VEL
LIN {X 0,Y 580.13,Z 713.597,A -85,B 0,C 180,E1 -1781.275,E2 -1781.275} C_VEL
LIN {X 0,Y 580.084,Z 718.732,A -85,B 0,C 180,E1 -1782.369,E2 -1782.369} C_VEL
LIN {X 0,Y 580.057,Z 721.715,A -85,B 0,C 180,E1 -1783.172,E2 -1783.172} C_VEL
LIN {X 0,Y 580.069,Z 723.655,A -85,B 0,C 180,E1 -1783.82,E2 -1783.82} C_VEL
LIN {X 0,Y 580.033,Z 725.383,A -85,B 0,C 180,E1 -1784.54,E2 -1784.54} C_VEL
LIN {X 0,Y 580.054,Z 727.295,A -85,B 0,C 180,E1 -1785.766,E2 -1785.766} C_VEL
LIN {X 0,Y 580.062,Z 727.926,A -85,B 0,C 180,E1 -1786.691,E2 -1786.691} C_VEL
LIN {X 0,Y 580.051,Z 727.925,A -85,B 0,C 180,E1 -1787.403,E2 -1787.403} C_VEL
LIN {X 0,Y 580.055,Z 727.527,A -85,B 0,C 180,E1 -1788.114,E2 -1788.114} C_VEL
LIN {X 0,Y 580.076,Z 726.528,A -85,B 0,C 180,E1 -1788.926,E2 -1788.926} C_VEL
LIN {X 0,Y 580.063,Z 723.753,A -85,B 0,C 180,E1 -1790.234,E2 -1790.234} C_VEL
LIN {X 0,Y 580.089,Z 720.39,A -85,B 0,C 180,E1 -1791.29,E2 -1791.29} C_VEL
LIN {X 0,Y 580.114,Z 715.975,A -85,B 0,C 180,E1 -1792.342,E2 -1792.342} C_VEL
LIN {X 0,Y 580.176,Z 710.463,A -85,B 0,C 180,E1 -1793.375,E2 -1793.375} C_VEL
LIN {X 0,Y 580.161,Z 703.342,A -85,B 0,C 180,E1 -1794.439,E2 -1794.439} C_VEL
LIN {X 0,Y 580.266,Z 694.654,A -85,B 0,C 180,E1 -1795.485,E2 -1795.485} C_VEL
LIN {X 0,Y 580.34,Z 684.761,A -85,B 0,C 180,E1 -1796.442,E2 -1796.442} C_VEL
LIN {X 0,Y 580.455,Z 674.755,A -85,B 0,C 180,E1 -1797.224,E2 -1797.224} C_VEL
LIN {X 0,Y 580.547,Z 663.751,A -85,B 0,C 180,E1 -1797.919,E2 -1797.919} C_VEL
LIN {X 0,Y 580.6,Z 651.357,A -85,B 0,C 180,E1 -1798.526,E2 -1798.526} C_VEL
LIN {X 0,Y 580.748,Z 639.501,A -85,B 0,C 180,E1 -1798.96,E2 -1798.96} C_VEL
LIN {X 0,Y 580.795,Z 625.548,A -85,B 0,C 180,E1 -1799.307,E2 -1799.307} C_VEL
LIN {X 0,Y 580.881,Z 590.855,A -85,B 0,C 180,E1 -1799.762,E2 -1799.762} C_VEL
LIN {X 0,Y 580.788,Z 518.746,A -85,B 0,C 180,E1 -1800.661,E2 -1800.661} C_VEL
LIN {X 0,Y 580.377,Z 515.902,A -85,B 0,C 180,E1 -1800.737,E2 -1800.737} C_VEL
LIN {X 0,Y 580.522,Z 498.942,A -85,B 0,C 180,E1 -1803.123,E2 -1803.123} C_VEL
LIN {X 0,Y 580.705,Z 478.435,A -85,B 0,C 180,E1 -1806.079,E2 -1806.079} C_VEL
LIN {X 0,Y 580.917,Z 458.174,A -85,B 0,C 180,E1 -1809.049,E2 -1809.049} C_VEL
LIN {X 0,Y 580.551,Z 453.512,A -85,B 0,C 180,E1 -1809.758,E2 -1809.758} C_VEL
LIN {X 0,Y 580.286,Z 452.293,A -85,B 0,C 180,E1 -1809.982,E2 -1809.982} C_VEL
LIN {X 0,Y 580.277,Z 452.201,A -85,B 0,C 180,E1 -1812.592,E2 -1812.592} C_VEL
LIN {X 0,Y 580.28,Z 452.203,A -85,B 0,C 180,E1 -1815.453,E2 -1815.453} C_VEL
LIN {X 0,Y 580.265,Z 452.202,A -85,B 0,C 180,E1 -1817.626,E2 -1817.626} C_VEL
LIN {X 0,Y 580.281,Z 452.198,A -85,B 0,C 180,E1 -1819.823,E2 -1819.823} C_VEL
LIN {X 0,Y 580.259,Z 452.2,A -85,B 0,C 180,E1 -1822.053,E2 -1822.053} C_VEL
LIN {X 0,Y 580.296,Z 452.203,A -85,B 0,C 180,E1 -1825.08,E2 -1825.08} C_VEL
LIN {X 0,Y 580.301,Z 452.196,A -85,B 0,C 180,E1 -1828.186,E2 -1828.186} C_VEL
LIN {X 0,Y 580.285,Z 452.205,A -85,B 0,C 180,E1 -1830.693,E2 -1830.693} C_VEL
LIN {X 0,Y 580.311,Z 452.195,A -85,B 0,C 180,E1 -1833.316,E2 -1833.316} C_VEL
LIN {X 0,Y 580.255,Z 452.201,A -85,B 0,C 180,E1 -1835.756,E2 -1835.756} C_VEL
LIN {X 0,Y 580.294,Z 452.199,A -85,B 0,C 180,E1 -1838.146,E2 -1838.146} C_VEL
LIN {X 0,Y 580.304,Z 452.2,A -85,B 0,C 180,E1 -1840.843,E2 -1840.843} C_VEL
LIN {X 0,Y 580.28,Z 452.198,A -85,B 0,C 180,E1 -1843.658,E2 -1843.658} C_VEL
LIN {X 0,Y 580.281,Z 452.204,A -85,B 0,C 180,E1 -1846.609,E2 -1846.609} C_VEL
LIN {X 0,Y 580.302,Z 452.195,A -85,B 0,C 180,E1 -1849.156,E2 -1849.156} C_VEL
LIN {X 0,Y 580.294,Z 452.198,A -85,B 0,C 180,E1 -1851.927,E2 -1851.927} C_VEL
LIN {X 0,Y 580.239,Z 452.208,A -85,B 0,C 180,E1 -1854.451,E2 -1854.451} C_VEL
LIN {X 0,Y 580.293,Z 452.197,A -85,B 0,C 180,E1 -1856.974,E2 -1856.974} C_VEL
LIN {X 0,Y 580.297,Z 452.197,A -85,B 0,C 180,E1 -1859.424,E2 -1859.424} C_VEL
LIN {X 0,Y 580.26,Z 452.208,A -85,B 0,C 180,E1 -1862.149,E2 -1862.149} C_VEL
LIN {X 0,Y 580.305,Z 452.412,A -85,B 0,C 180,E1 -1862.964,E2 -1862.964} C_VEL
LIN {X 0,Y 581.614,Z 457.736,A -85,B 0,C 180,E1 -1863.642,E2 -1863.642} C_VEL
LIN {X 0,Y 581.435,Z 477.927,A -85,B 0,C 180,E1 -1865.923,E2 -1865.923} C_VEL
LIN {X 0,Y 581.165,Z 502.236,A -85,B 0,C 180,E1 -1868.616,E2 -1868.616} C_VEL
LIN {X 0,Y 580.907,Z 528.559,A -85,B 0,C 180,E1 -1871.482,E2 -1871.482} C_VEL
LIN {X 0,Y 580.598,Z 553.875,A -85,B 0,C 180,E1 -1874.194,E2 -1874.194} C_VEL
LIN {X 0,Y 580.523,Z 573.848,A -85,B 0,C 180,E1 -1876.299,E2 -1876.299} C_VEL
LIN {X 0,Y 580.981,Z 579.633,A -85,B 0,C 180,E1 -1876.4,E2 -1876.4} C_VEL
LIN {X 0,Y 580.803,Z 683.89,A -85,B 0,C 180,E1 -1877.707,E2 -1877.707} C_VEL
LIN {X 0,Y 580.735,Z 697.182,A -85,B 0,C 180,E1 -1878.016,E2 -1878.016} C_VEL
LIN {X 0,Y 580.66,Z 709.345,A -85,B 0,C 180,E1 -1878.435,E2 -1878.435} C_VEL
LIN {X 0,Y 580.563,Z 721.611,A -85,B 0,C 180,E1 -1879.008,E2 -1879.008} C_VEL
LIN {X 0,Y 580.448,Z 733.186,A -85,B 0,C 180,E1 -1879.711,E2 -1879.711} C_VEL
LIN {X 0,Y 580.344,Z 743.585,A -85,B 0,C 180,E1 -1880.502,E2 -1880.502} C_VEL
LIN {X 0,Y 580.267,Z 752.101,A -85,B 0,C 180,E1 -1881.291,E2 -1881.291} C_VEL
LIN {X 0,Y 580.223,Z 759.951,A -85,B 0,C 180,E1 -1882.167,E2 -1882.167} C_VEL
LIN {X 0,Y 580.155,Z 767.644,A -85,B 0,C 180,E1 -1883.221,E2 -1883.221} C_VEL
LIN {X 0,Y 580.139,Z 774.674,A -85,B 0,C 180,E1 -1884.437,E2 -1884.437} C_VEL
LIN {X 0,Y 580.108,Z 779.367,A -85,B 0,C 180,E1 -1885.482,E2 -1885.482} C_VEL
LIN {X 0,Y 580.123,Z 782.953,A -85,B 0,C 180,E1 -1886.526,E2 -1886.526} C_VEL
LIN {X 0,Y 580.043,Z 784.806,A -85,B 0,C 180,E1 -1887.221,E2 -1887.221} C_VEL
LIN {X 0,Y 580.039,Z 786.198,A -85,B 0,C 180,E1 -1887.916,E2 -1887.916} C_VEL
LIN {X 0,Y 580.04,Z 787.784,A -85,B 0,C 180,E1 -1889.305,E2 -1889.305} C_VEL
LIN {X 0,Y 580.037,Z 788,A -85,B 0,C 180,E1 -1889.999,E2 -1889.999} C_VEL
LIN {X 0,Y 580.046,Z 787.187,A -85,B 0,C 180,E1 -1891.387,E2 -1891.387} C_VEL
LIN {X 0,Y 580.039,Z 786.203,A -85,B 0,C 180,E1 -1892.082,E2 -1892.082} C_VEL
LIN {X 0,Y 580.043,Z 784.813,A -85,B 0,C 180,E1 -1892.777,E2 -1892.777} C_VEL
LIN {X 0,Y 580.11,Z 781.9,A -85,B 0,C 180,E1 -1893.819,E2 -1893.819} C_VEL
LIN {X 0,Y 580.053,Z 777.954,A -85,B 0,C 180,E1 -1894.864,E2 -1894.864} C_VEL
LIN {X 0,Y 580.139,Z 771.884,A -85,B 0,C 180,E1 -1896.084,E2 -1896.084} C_VEL
LIN {X 0,Y 580.184,Z 765.246,A -85,B 0,C 180,E1 -1897.131,E2 -1897.131} C_VEL
LIN {X 0,Y 580.25,Z 757.001,A -85,B 0,C 180,E1 -1898.181,E2 -1898.181} C_VEL
LIN {X 0,Y 580.307,Z 748.551,A -85,B 0,C 180,E1 -1899.057,E2 -1899.057} C_VEL
LIN {X 0,Y 580.418,Z 738.113,A -85,B 0,C 180,E1 -1899.935,E2 -1899.935} C_VEL
LIN {X 0,Y 580.515,Z 727.778,A -85,B 0,C 180,E1 -1900.638,E2 -1900.638} C_VEL
LIN {X 0,Y 580.596,Z 716.252,A -85,B 0,C 180,E1 -1901.264,E2 -1901.264} C_VEL
LIN {X 0,Y 580.668,Z 703.509,A -85,B 0,C 180,E1 -1901.784,E2 -1901.784} C_VEL
LIN {X 0,Y 580.747,Z 690.489,A -85,B 0,C 180,E1 -1902.159,E2 -1902.159} C_VEL
LIN {X 0,Y 580.856,Z 678.178,A -85,B 0,C 180,E1 -1902.378,E2 -1902.378} C_VEL
LIN {X 0,Y 580.828,Z 576.248,A -85,B 0,C 180,E1 -1903.646,E2 -1903.646} C_VEL
LIN {X 0,Y 580.519,Z 573.588,A -85,B 0,C 180,E1 -1903.721,E2 -1903.721} C_VEL
LIN {X 0,Y 580.742,Z 547.279,A -85,B 0,C 180,E1 -1906.521,E2 -1906.521} C_VEL
LIN {X 0,Y 580.934,Z 521.305,A -85,B 0,C 180,E1 -1909.33,E2 -1909.33} C_VEL
LIN {X 0,Y 581.235,Z 495.168,A -85,B 0,C 180,E1 -1912.2,E2 -1912.2} C_VEL
LIN {X 0,Y 581.583,Z 469.953,A -85,B 0,C 180,E1 -1915.019,E2 -1915.019} C_VEL
LIN {X 0,Y 581.679,Z 458.087,A -85,B 0,C 180,E1 -1916.371,E2 -1916.371} C_VEL
LIN {X 0,Y 580.269,Z 452.272,A -85,B 0,C 180,E1 -1917.133,E2 -1917.133} C_VEL
LIN {X 0,Y 580.259,Z 452.207,A -85,B 0,C 180,E1 -1919.773,E2 -1919.773} C_VEL
LIN {X 0,Y 580.29,Z 452.206,A -85,B 0,C 180,E1 -1922.199,E2 -1922.199} C_VEL
LIN {X 0,Y 580.269,Z 452.201,A -85,B 0,C 180,E1 -1924.696,E2 -1924.696} C_VEL
LIN {X 0,Y 580.263,Z 452.199,A -85,B 0,C 180,E1 -1927.269,E2 -1927.269} C_VEL
LIN {X 0,Y 580.278,Z 452.206,A -85,B 0,C 180,E1 -1930.268,E2 -1930.268} C_VEL
LIN {X 0,Y 580.263,Z 452.201,A -85,B 0,C 180,E1 -1932.706,E2 -1932.706} C_VEL
LIN {X 0,Y 580.246,Z 452.202,A -85,B 0,C 180,E1 -1935.609,E2 -1935.609} C_VEL
LIN {X 0,Y 580.262,Z 452.202,A -85,B 0,C 180,E1 -1938.669,E2 -1938.669} C_VEL
LIN {X 0,Y 580.258,Z 452.2,A -85,B 0,C 180,E1 -1940.963,E2 -1940.963} C_VEL
LIN {X 0,Y 580.236,Z 452.203,A -85,B 0,C 180,E1 -1943.594,E2 -1943.594} C_VEL
